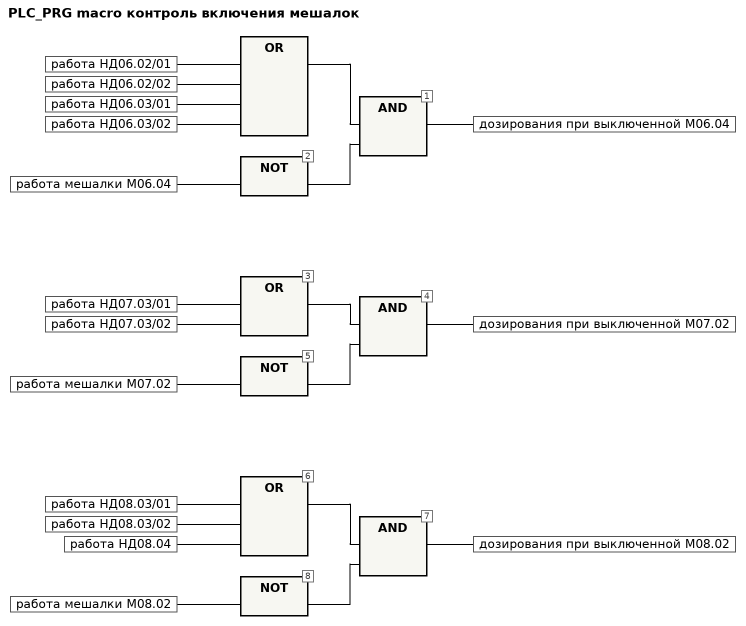
[picture p24: PLC_PRG macro контроль включения мешалок (CFC)]
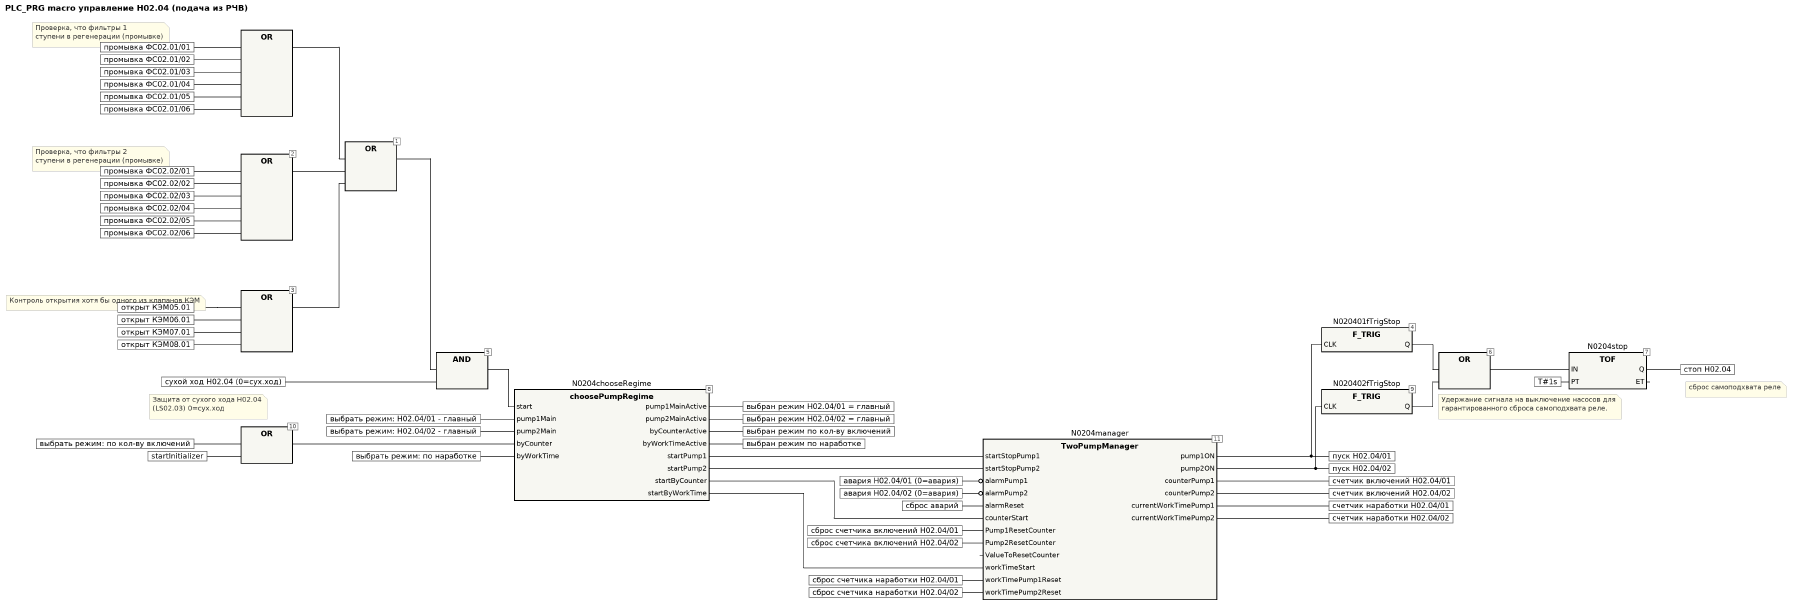
_CFC_ (* Continuous Function Chart, elements in execution order *)
(* Пуск Н02.04/02 *)
(* Пуск Н02.04/01 *)
(* Стоп Н02.04 *)
(* Сухой ход Н02.04 (LS02.03) 0=сух.ход *)
(* Клапан КЭМ08.01 открыт. *)
(* Клапан КЭМ07.01 открыт. *)
(* Клапан КЭМ06.01 открыт. *)
(* Клапан КЭМ05.01 открыт. *)
(* промывка ФС02.02/01 *)
(* промывка ФС02.02/02 *)
(* промывка ФС02.02/03 *)
(* промывка ФС02.02/04 *)
(* промывка ФС02.02/05 *)
(* промывка ФС02.02/06 *)
(* Авария Н02.04/02 (0=авария) *)
(* Авария Н02.04/01 (0=авария) *)
(* импульсный расходомер *)
(* авария Н04.04/02, 0=авария *)
(* авария Н04.04/01, 0=авария *)
(* сухой ход Н04.04, 0=защита *)
(* авт.пуск Н04.04 *)
(* пуск Н04.04/01 *)
(* пуск Н04.04/02 *)
(* стоп Н04.04 *)
(* подающий насос ФПК работает *)
(* статус КШЭ04.01 закрыт *)
(* Закрыть КШЭ04.01 *)
(* статус КШЭ04.01 открыт *)
(* Открыть КШЭ04.01 *)
(* авария ФПК *)
(* Авария входа AI6 ПЛК, давл.ФПК *)
(* Давление на входе ФПК / 0...16 бар (мах допуст.10) *)
(* LSА02.01 Перелив РЧВ02.03 *)
(* авария питания ЗДЭ02.25 *)
(* термоконтакт Н01.05/02 *)
(* термоконтакт Н01.05/01 *)
(* Авария ЧРП Н01.05 *)
(* КМ3 питание насоса 2 *)
(* КМ2 питание насоса 1 *)
(* КМ1 питание ЧРП *)
(* Пуск  Н01.05 *)
(* время на создание потока *)
(* управление Н01.05 - поддержание заданного расхода по FT01.02 *)
(* Стоп  Н01.05 (сброс самоподхвата реле) *)
(* SA1 Ручной выбор Н01.05/02 = главный *)
(* SA1 Ручной выбор Н01.05/01 = главный *)
(* LS01.04 - нижний уровень ОГМ01.04, сухой ход Н01.05 *)
(* LS01.03 - рабочий верхний уровень ОГМ01.04 автоматический пуск 01.05 *)
(* Статус ПУСК ЧРП Н01.05 *)
(* Инициализирует требуемые булевые переменные / в момент старта выполнения программы. *)
(* LSA01.02 перелив ОГМ01.04 *)
(* сухой ход НД08.03/02 *)
(* сухой ход НД08.03/01 *)
(* сухой ход НД08.03/02 *)
(* сухой ход НД08.03/01 *)
(* авария входа рН-метра QE01.02 *)
(* рН-метр QE01.01 на входе, / диапазон 0...14 *)
(* расходомер FT01.02 на входе, / диапазон 0...600куб/час *)
(* авария входа расходомера FT01.01 *)
(* управление 4...20мА НД08.04 *)
(* пуск/стоп НД08.04 *)
(* насос Н04.01 работает *)
(* авария НД08.04 *)
(* авария привода НД08.03/02 *)
(* авария привода НД08.03/01 *)
(* АВАРИИ *)
(* управление 4...20мА НД05.02/02 *)
(* пуск/стоп НД05.02/02 *)
(* авария НД05.02/02 *)
(* авария НД05.02/01 *)
(* пуск/стоп НД05.02/01 *)
(* управление 4...20мА НД05.02/01 *)
(* датчик температуры в помещении / (метран) диапазон: 0...+100С *)
(* лампа АВАРИЯ *)
(* авария входа датчика температуры *)
(* ошибка блока дозирования НД05.02 *)
(* авария НД06.02/02 *)
(* авария НД06.02/01 *)
(* управление 4...20мА НД06.02/02 *)
(* пуск/стоп НД06.02/02 *)
(* пуск/стоп НД06.02/01 *)
(* управление 4...20мА НД06.02/01 *)
(* авария НД06.03/02 *)
(* авария НД06.03/01 *)
(* управление 4...20мА НД06.03/02 *)
(* пуск/стоп НД06.03/02 *)
(* пуск/стоп НД06.03/01 *)
(* управление 4...20мА НД06.03/01 *)
(* авария НД05.02/02 *)
(* авария НД05.02/01 *)
(* авария НД06.02/02 *)
(* авария НД06.02/01 *)
(* авария НД06.03/02 *)
(* авария НД06.03/01 *)
(* авария НД07.03/02 *)
(* авария НД07.03/01 *)
(* пуск/стоп НД07.03/02 *)
(* пуск/стоп НД07.03/01 *)
(* управление 4...20мА НД07.03/02 *)
(* управление 4...20мА НД07.03/01 *)
(* авария НД07.03/02 *)
(* авария НД07.03/01 *)
(* авария привода НД08.03/02 *)
(* авария привода НД08.03/01 *)
(* управление 4...20мА НД08.03/02 *)
(* пуск/стоп НД08.03/02 *)
(* пуск/стоп НД08.03/01 *)
(* управление 4...20мА НД08.03/01 *)
(* авария НД08.04 *)
(* расходомер FT01.01 на входе, / диапазон 0...600куб/час *)
(* авария входа расходомера FT01.02 *)
(* авария входа рН-метра QE01.01 *)
(* рН-метр QE01.02 на входе, / диапазон 0...14 *)
(* статус ЗДЭ02.25 закрыт *)
(* LS02.02 Раб.верх.уровень РЧВ02.03 *)
(* Закрыть ЗДЭ02.25 *)
(* статус ЗДЭ02.25 открыт *)
(* LSА02.01 Перелив РЧВ02.03 *)
(* Открыть ЗДЭ02.25 *)
(* ФПК не запустился *)
(* ФПК готов к приему *)
(* подающий насос ФПК работает *)
(* авария ФПК *)
(* Давление на входе ФПК (0...16 бар) *)
(* датчик уровня осадка *)
(* Защита от сухого хода насоса ФПК *)
(* запуск фильтрации *)
(* время работы ФПК после спада сигнала датч.осадка *)
(* время контроля старта ФПК (по умолч.=3мин) *)
(* авария Н04.04/02 *)
(* авария Н04.04/01 *)
(* УФО вкл вручную без потока *)
(* авария УФО03.01/01 *)
(* авария УФО03.01/02 *)
(* авт.пускУФО03.01/01 *)
(* работа УФО03.01/01 *)
(* Для подачи предостережения на пульте / оператора (при необходимости), а также / сигнализации лампой АВАРИЯ. *)
(* авт.пускУФО03.01/02 *)
(* авария УФО03.01/01 *)
(* работа УФО03.01/02 *)
(* авария УФО03.01/02 *)
(* Контроль, если УФО включили вручную, / а потока при этом нет. *)
(* работа М06.04 (УПК) *)
(* работа М07.02 (УПЩ) *)
(* работа М08.02 (УПФ) *)
(* авария М06.04 (УПК) *)
(* авария М07.02 (УПЩ) *)
(* авария М08.02 (УПФ) *)
(* пуск/стоп НД07.03/02 *)
(* пуск/стоп НД07.03/01 *)
(* пуск/стоп НД08.04 *)
(* пуск/стоп НД06.02/02 *)
(* пуск/стоп НД06.02/01 *)
(* пуск/стоп НД06.03/02 *)
(* пуск/стоп НД06.03/01 *)
(* пуск/стоп НД08.03/02 *)
(* пуск/стоп НД08.03/01 *)
(* Авария Н02.04/02 (0=авария) *)
(* Защита от сухого хода Н02.04 / (LS02.03) 0=сух.ход *)
(* Авария Н02.04/01 (0=авария) *)
(* Стоп Н02.04 *)
(* Пуск Н02.04/02 *)
(* Пуск Н02.04/01 *)
(* Контроль открытия хотя бы одного из клапанов КЭМ *)
(* Клапан КЭМ08.01 открыт. *)
(* Клапан КЭМ07.01 открыт. *)
(* Клапан КЭМ06.01 открыт. *)
(* Клапан КЭМ05.01 открыт. *)
(* Удержание сигнала на выключение насосов для / гарантированного сброса самоподхвата реле. *)
(* промывка ФС02.02/01 *)
(* Проверка, что фильтры 2 / ступени в регенерации (промывке) *)
(* промывка ФС02.02/02 *)
(* промывка ФС02.02/03 *)
(* промывка ФС02.02/04 *)
(* промывка ФС02.02/05 *)
(* промывка ФС02.02/06 *)
(* промывка ФС02.01/01 *)
(* Проверка, что фильтры 1 / ступени в регенерации (промывке) *)
(* промывка ФС02.01/02 *)
(* промывка ФС02.01/03 *)
(* промывка ФС02.01/04 *)
(* промывка ФС02.01/05 *)
(* промывка ФС02.01/06 *)
(* промывка ФС02.01/01 *)
(* промывка ФС02.01/02 *)
(* промывка ФС02.01/03 *)
(* промывка ФС02.01/04 *)
(* промывка ФС02.01/05 *)
(* промывка ФС02.01/06 *)
(* Авария Н02.04/02 (0=авария) *)
(* Авария Н02.04/01 (0=авария) *)
#0 rTrigStartInitializer:R_TRIG(CLK: TRUE)
#1 startInitializer <= #0.Q
#2 MACRO контроль аналогового входа DD1_AI1(pin 1 "вход": DD1_AI1)
	(* Не смотрим конкретную ошибку, / определяем,что вход неисправен без расшифровки. *)
	#3 DD1_AI1_FT0101:DECODE_FLOAT(VALUE: pin 1, DEF_VALUE: -)
	#4 NE(#3._ERR, 0)
	out 2 "авария" <= #4
	out 1 "выход" <= #3.OUT_VALUE
END_MACRO
#5 DD1_AI1_FT0101value <= #2.out 1
#6 DD1_AI1_error <= #2.out 2
#7 MACRO контроль аналогового входа DD1_AI2(pin 1 "вход": DD1_AI2)
	(* Не смотрим конкретную ошибку, / определяем,что вход неисправен без расшифровки. *)
	#8 DD1_AI2_FT0102:DECODE_FLOAT(VALUE: pin 1, DEF_VALUE: -)
	#9 NE(#8._ERR, 0)
	out 2 "авария" <= #9
	out 1 "выход" <= #8.OUT_VALUE
END_MACRO
#10 DD1_AI2_FT0102value <= #7.out 1
#11 DD1_AI2_error <= #7.out 2
#12 MACRO контроль аналогового входа DD1_AI3(pin 1 "вход": DD1_AI3)
	(* Не смотрим конкретную ошибку, / определяем,что вход неисправен без расшифровки. *)
	#13 DD1_AI3_QE0101:DECODE_FLOAT(VALUE: pin 1, DEF_VALUE: -)
	#14 NE(#13._ERR, 0)
	out 2 "авария" <= #14
	out 1 "выход" <= #13.OUT_VALUE
END_MACRO
#15 DD1_AI3_QE0101value <= #12.out 1
#16 DD1_AI3_error <= #12.out 2
#17 OR(DD1_AI0_error, alarmHighTemperature, alarmLowTemperature, ND0502dosingError, NOT DD6_DI.0, NOT DD6_DI.1, ND0502dosingError, NOT DD6_DI.2, NOT DD6_DI.3, ND0602dosingError, NOT DD6_DI.4, NOT DD6_DI.5, ND0603dosingError, NOT DD6_DI.6, NOT DD6_DI.7, ND0803dosingError, NOT DD5_DI.12, NOT DD5_DI.13, DD1_DI6, DD1_DI7, NOT DD6_DI.16, ND0804dosingError, DD1_AI1_error, DD1_AI2_error, DD1_AI3_error, DD1_AI4_error, NOT DD6_DI.11, N010501alarm, N010502alarm, NOT DD9_DI.28, ZDE0225errorToOpen, ZDE0225errorToClose, NOT DD6_DI.13, DD1_AI5_error, DD7_DI.14, FPKnotStarted, FPKneedToClean, FPKkshe0401errorToOpen, FPKkshe0401errorToClose, NOT DD5_DI.14, NOT DD5_DI.15, DD5_DI.27, DD5_DI.29, UFO0301noFlowAttention, NOT DD5_DI.20, NOT DD5_DI.22, NOT DD5_DI.24, NOT DD5_DI.7, NOT DD5_DI.8)
#18 DD1_DO11 <= #17
#19 MACRO управление НД06.02 УПК(pin 1 "вход расходомера в куб/час": DD1_AI2_FT0102value, pin 2 "max производительность НД в мл/мин": ND0602setMaxDosVal, pin 3 "задание дозирования в мл/куб": ND0602setKoefProp, pin 4 "режим:1 насос главный": ND0602regimeP1M, pin 5 "режим: 2 насос главный": ND0602regimeP2M, pin 6 "режим: по наработке": ND0602regimeByWT, pin 7 "режим: по кол-ву включений": ND0602regimeByC, pin 8 "авария 1 насоса": DD6_DI.2, pin 9 "авария 2 насоса": DD6_DI.3, pin 10 "сброс аварий": alarmReset, pin 11 "сброс счетчика включений 1 насоса": ND0602resetCountP1, pin 12 "сброс ссчетчика включений 2 насоса": ND0602resetCountP2, pin 13 "сброс наработки 1 насоса": ND0602resetWorkTimeP1, pin 14 "сброс наработки 2 насоса": ND0602resetWorkTimeP2)
	(* Если на входе SEL = TRUE, / то нижнее значение, / иначе - то,что посередине. *)
	(* сигнал 4...20мА на НД06.02/01 *)
	(* сигнал 4...20мА на НД06.02/02 *)
	#20 SEL(#27.pump1ON, 0, #22.outputValue)
	#21 REAL_TO_WORD(#20)
	out 6 "выход 4...20мА насоса 1" <= #21
	#22 ND0602dosing:DosingPumpProportional(flowValue: pin 1, setMinPumpDosingValue: -, setMaxPumpDosingValue: pin 2, minOutputValue: -, maxOutputValue: -, setKoeffProportionality: pin 3, minFlowToStart: -)
	out 1 "ошибка блока дозирования" <= #22.dosingError
	#23 SEL(#27.pump2ON, 0, #22.outputValue)
	#24 REAL_TO_WORD(#23)
	out 7 "выход 4...20мА насоса 2" <= #24
	#25 ND0602regime:choosePumpRegime(start: #22.startDosingPump, pump1Main: pin 4, pump2Main: pin 5, byCounter: #26, byWorkTime: pin 6)
	out 2 "статус: 1 насос главный" <= #25.pump1MainActive
	out 3 "статус: 2 насос главный" <= #25.pump2MainActive
	out 4 "статус: по кол-ву включений" <= #25.byCounterActive
	#26 OR(pin 7, startInitializer)
	out 5 "статус: по наработке" <= #25.byWorkTimeActive
	#27 ND0602manager:TwoPumpManager(startStopPump1: #25.startPump1, startStopPump2: #25.startPump2, alarmPump1: #28, alarmPump2: #29, alarmReset: pin 10, counterStart: #25.startByCounter, Pump1ResetCounter: pin 11, Pump2ResetCounter: pin 12, ValueToResetCounter: -, workTimeStart: #25.startByWorkTime, workTimePump1Reset: pin 13, workTimePump2Reset: pin 14)
	out 12 "сигнал на включение насоса 1" <= #27.pump1ON
	#28 NOT(pin 8)
	out 13 "сигнал на включение насоса 2" <= #27.pump2ON
	out 8 "счетчик включений насоса 1" <= #27.counterPump1
	#29 NOT(pin 9)
	out 9 "счетчик включений насоса 2" <= #27.counterPump2
	out 10 "счетчик наработки насоса 1" <= #27.currentWorkTimePump1
	out 11 "счетчик наработки насоса 2" <= #27.currentWorkTimePump2
END_MACRO
#30 ND0602dosingError <= #19.out 1
#31 ND0602statRegimeP1M <= #19.out 2
#32 ND0602statRegimeP2M <= #19.out 3
#33 ND0602statRegimeByC <= #19.out 4
#34 ND0602statRegimeByWT <= #19.out 5
#35 DD10_AO1 <= #19.out 6
#36 DD10_AO2 <= #19.out 7
#37 ND0602counterP1 <= #19.out 8
#38 ND0602counterP2 <= #19.out 9
#39 ND0602workTimeP1 <= #19.out 10
#40 ND0602workTimeP2 <= #19.out 11
#41 DD4_DO.6 <= #19.out 12
#42 DD4_DO.7 <= #19.out 13
#43 MACRO контроль аналогового входа DD1_AI4(pin 1 "вход": DD1_AI4)
	(* Не смотрим конкретную ошибку, / определяем,что вход неисправен без расшифровки. *)
	#44 DD1_AI4_QE0102:DECODE_FLOAT(VALUE: pin 1, DEF_VALUE: -)
	#45 NE(#44._ERR, 0)
	out 2 "авария" <= #45
	out 1 "выход" <= #44.OUT_VALUE
END_MACRO
#46 DD1_AI4_QE0102value <= #43.out 1
#47 DD1_AI4_error <= #43.out 2
#48 MACRO управление НД05.02 УПГ(pin 1 "вход расходомера в куб/час": DD1_AI1_FT0101value, pin 2 "max производительность НД в мл/мин": ND0502setMaxDosVal, pin 3 "задание дозирования в мл/куб": ND0502setKoefProp, pin 4 "режим:1 насос главный": ND0502regimeP1M, pin 5 "режим: 2 насос главный": ND0502regimeP2M, pin 6 "режим: по наработке": ND0502regimeByWT, pin 7 "режим: по кол-ву включений": ND0502regimeByC, pin 8 "авария 1 насоса": DD6_DI.0, pin 9 "авария 2 насоса": DD6_DI.1, pin 10 "сброс аварий": alarmReset, pin 11 "сброс счетчика включений 1 насоса": ND0502resetCountP1, pin 12 "сброс ссчетчика включений 2 насоса": ND0502resetCountP2, pin 13 "сброс наработки 1 насоса": ND0502resetWorkTimeP1, pin 14 "сброс наработки 2 насоса": ND0502resetWorkTimeP2)
	(* Если на входе SEL = TRUE, / то нижнее значение, / иначе - то,что посередине. *)
	(* сигнал 4...20мА на НД05.02/01 *)
	(* сигнал 4...20мА на НД05.02/02 *)
	#49 SEL(#55.pump1ON, 0, #50.outputValue)
	out 6 "выход 4...20мА насоса 1" <= #49
	#50 ND0502dosing:DosingPumpProportional(flowValue: pin 1, setMinPumpDosingValue: -, setMaxPumpDosingValue: pin 2, minOutputValue: -, maxOutputValue: -, setKoeffProportionality: pin 3, minFlowToStart: -)
	out 1 "ошибка блока дозирования" <= #50.dosingError
	#51 SEL(#55.pump2ON, 0, #50.outputValue)
	#52 REAL_TO_WORD(#51)
	out 7 "выход 4...20мА насоса 2" <= #52
	#53 ND0502regime:choosePumpRegime(start: #50.startDosingPump, pump1Main: pin 4, pump2Main: pin 5, byCounter: #54, byWorkTime: pin 6)
	out 2 "статус: 1 насос главный" <= #53.pump1MainActive
	out 3 "статус: 2 насос главный" <= #53.pump2MainActive
	out 4 "статус: по кол-ву включений" <= #53.byCounterActive
	#54 OR(pin 7, startInitializer)
	out 5 "статус: по наработке" <= #53.byWorkTimeActive
	#55 ND0502manager:TwoPumpManager(startStopPump1: #53.startPump1, startStopPump2: #53.startPump2, alarmPump1: #56, alarmPump2: #57, alarmReset: pin 10, counterStart: #53.startByCounter, Pump1ResetCounter: pin 11, Pump2ResetCounter: pin 12, ValueToResetCounter: -, workTimeStart: #53.startByWorkTime, workTimePump1Reset: pin 13, workTimePump2Reset: pin 14)
	out 12 "сигнал на включение насоса 1" <= #55.pump1ON
	#56 NOT(pin 8)
	out 13 "сигнал на включение насоса 2" <= #55.pump2ON
	out 8 "счетчик включений насоса 1" <= #55.counterPump1
	#57 NOT(pin 9)
	out 9 "счетчик включений насоса 2" <= #55.counterPump2
	out 10 "счетчик наработки насоса 1" <= #55.currentWorkTimePump1
	out 11 "счетчик наработки насоса 2" <= #55.currentWorkTimePump2
END_MACRO
#58 ND0502dosingError <= #48.out 1
#59 ND0502statRegimeP1M <= #48.out 2
#60 ND0502statRegimeP2M <= #48.out 3
#61 ND0502statRegimeByC <= #48.out 4
#62 ND0502statRegimeByWT <= #48.out 5
#63 DD1_AO3 <= #48.out 6
#64 DD10_AO0 <= #48.out 7
#65 ND0502counterP1 <= #48.out 8
#66 ND0502counterP2 <= #48.out 9
#67 ND0502workTimeP1 <= #48.out 10
#68 ND0502workTimeP2 <= #48.out 11
#69 DD4_DO.4 <= #48.out 12
#70 DD4_DO.5 <= #48.out 13
#71 MACRO управление НД06.03 УПК(pin 1 "вход расходомера в куб/час": DD1_AI1_FT0101value, pin 2 "max производительность НД в мл/мин": ND0603setMaxDosVal, pin 3 "задание дозирования в мл/куб": ND0603setKoefProp, pin 4 "режим:1 насос главный": ND0603regimeP1M, pin 5 "режим: 2 насос главный": ND0603regimeP2M, pin 6 "режим: по наработке": ND0603regimeByWT, pin 7 "режим: по кол-ву включений": ND0603regimeByC, pin 8 "авария 1 насоса": DD6_DI.4, pin 9 "авария 2 насоса": DD6_DI.5, pin 10 "сброс аварий": alarmReset, pin 11 "сброс счетчика включений 1 насоса": ND0603resetCountP1, pin 12 "сброс ссчетчика включений 2 насоса": ND0603resetCountP2, pin 13 "сброс наработки 1 насоса": ND0603resetWorkTimeP1, pin 14 "сброс наработки 2 насоса": ND0603resetWorkTimeP2)
	(* Если на входе SEL = TRUE, / то нижнее значение, / иначе - то,что посередине. *)
	(* сигнал 4...20мА на НД06.03/01 *)
	(* сигнал 4...20мА на НД06.03/02 *)
	#72 SEL(#79.pump1ON, 0, #74.outputValue)
	#73 REAL_TO_WORD(#72)
	out 6 "выход 4...20мА насоса 1" <= #73
	#74 ND0603dosing:DosingPumpProportional(flowValue: pin 1, setMinPumpDosingValue: -, setMaxPumpDosingValue: pin 2, minOutputValue: -, maxOutputValue: -, setKoeffProportionality: pin 3, minFlowToStart: -)
	out 1 "ошибка блока дозирования" <= #74.dosingError
	#75 SEL(#79.pump2ON, 0, #74.outputValue)
	#76 REAL_TO_WORD(#75)
	out 7 "выход 4...20мА насоса 2" <= #76
	#77 ND0603regime:choosePumpRegime(start: #74.startDosingPump, pump1Main: pin 4, pump2Main: pin 5, byCounter: #78, byWorkTime: pin 6)
	out 2 "статус: 1 насос главный" <= #77.pump1MainActive
	out 3 "статус: 2 насос главный" <= #77.pump2MainActive
	out 4 "статус: по кол-ву включений" <= #77.byCounterActive
	#78 OR(pin 7, startInitializer)
	out 5 "статус: по наработке" <= #77.byWorkTimeActive
	#79 ND0603manager:TwoPumpManager(startStopPump1: #77.startPump1, startStopPump2: #77.startPump2, alarmPump1: #80, alarmPump2: #81, alarmReset: pin 10, counterStart: #77.startByCounter, Pump1ResetCounter: pin 11, Pump2ResetCounter: pin 12, ValueToResetCounter: -, workTimeStart: #77.startByWorkTime, workTimePump1Reset: pin 13, workTimePump2Reset: pin 14)
	out 12 "сигнал на включение насоса 1" <= #79.pump1ON
	#80 NOT(pin 8)
	out 13 "сигнал на включение насоса 2" <= #79.pump2ON
	out 8 "счетчик включений насоса 1" <= #79.counterPump1
	#81 NOT(pin 9)
	out 9 "счетчик включений насоса 2" <= #79.counterPump2
	out 10 "счетчик наработки насоса 1" <= #79.currentWorkTimePump1
	out 11 "счетчик наработки насоса 2" <= #79.currentWorkTimePump2
END_MACRO
#82 ND0603dosingError <= #71.out 1
#83 ND0603statRegimeP1M <= #71.out 2
#84 ND0603statRegimeP2M <= #71.out 3
#85 ND0603statRegimeByC <= #71.out 4
#86 ND0603statRegimeByWT <= #71.out 5
#87 DD10_AO3 <= #71.out 6
#88 DD10_AO4 <= #71.out 7
#89 ND0603counterP1 <= #71.out 8
#90 ND0603counterP2 <= #71.out 9
#91 ND0603workTimeP1 <= #71.out 10
#92 ND0603workTimeP2 <= #71.out 11
#93 DD4_DO.8 <= #71.out 12
#94 DD4_DO.9 <= #71.out 13
#95 MACRO управление НД08.03 УПФ(pin 1 "вход расходомера в куб/час": DD1_AI1_FT0101value, pin 2 "max производительность НД в мл/мин": ND0803setMaxDosVal, pin 3 "задание дозирования в мл/куб": ND0803setKoefProp, pin 4 "режим:1 насос главный": ND0803regimeP1M, pin 5 "режим: 2 насос главный": ND0803regimeP2M, pin 6 "режим: по наработке": ND0803regimeByWT, pin 7 "режим: по кол-ву включений": ND0803regimeByC, pin 8 "авария 1 насоса": DD5_DI.12, pin 9 "авария 2 насоса": DD5_DI.13, pin 10 "сброс аварий": alarmReset, pin 11 "сброс счетчика включений 1 насоса": ND0803resetCountP1, pin 12 "сброс ссчетчика включений 2 насоса": ND0803resetCountP2, pin 13 "сброс наработки 1 насоса": ND0803resetWorkTimeP1, pin 14 "сброс наработки 2 насоса": ND0803resetWorkTimeP2, pin 15 "сухой ход 1 насоса": DD1_DI6, pin 16 "сухой ход 2 насоса": DD1_DI7)
	(* Если на входе SEL = TRUE, / то нижнее значение, / иначе - то,что посередине. *)
	(* сигнал 4...20мА на НД08.03/01 *)
	(* сигнал 4...20мА на НД08.03/02 *)
	#96 SEL(#105.pump1ON, 0, #97.outputValue)
	out 6 "выход 4...20мА насоса 1" <= #96
	#97 ND0803dosing:DosingPumpProportional(flowValue: pin 1, setMinPumpDosingValue: -, setMaxPumpDosingValue: pin 2, minOutputValue: -, maxOutputValue: -, setKoeffProportionality: pin 3, minFlowToStart: -)
	out 1 "ошибка блока дозирования" <= #97.dosingError
	#98 SEL(#105.pump2ON, 0, #97.outputValue)
	out 7 "выход 4...20мА насоса 2" <= #98
	#99 ND0803regime:choosePumpRegime(start: #97.startDosingPump, pump1Main: pin 4, pump2Main: pin 5, byCounter: #100, byWorkTime: pin 6)
	out 2 "статус: 1 насос главный" <= #99.pump1MainActive
	out 3 "статус: 2 насос главный" <= #99.pump2MainActive
	out 4 "статус: по кол-ву включений" <= #99.byCounterActive
	#100 OR(pin 7, startInitializer)
	out 5 "статус: по наработке" <= #99.byWorkTimeActive
	out 12 "сигнал на включение насоса 1" <= #105.pump1ON
	#101 NOT(pin 8)
	#102 OR(#101, pin 15)
	out 13 "сигнал на включение насоса 2" <= #105.pump2ON
	#103 NOT(pin 9)
	#104 OR(#103, pin 16)
	#105 ND0803manager:TwoPumpManager(startStopPump1: #99.startPump1, startStopPump2: #99.startPump2, alarmPump1: #102, alarmPump2: #104, alarmReset: pin 10, counterStart: #99.startByCounter, Pump1ResetCounter: pin 11, Pump2ResetCounter: pin 12, ValueToResetCounter: -, workTimeStart: #99.startByWorkTime, workTimePump1Reset: pin 13, workTimePump2Reset: pin 14)
	out 8 "счетчик включений насоса 1" <= #105.counterPump1
	out 9 "счетчик включений насоса 2" <= #105.counterPump2
	out 10 "счетчик наработки насоса 1" <= #105.currentWorkTimePump1
	out 11 "счетчик наработки насоса 2" <= #105.currentWorkTimePump2
END_MACRO
#106 ND0803dosingError <= #95.out 1
#107 ND0803statRegimeP1M <= #95.out 2
#108 ND0803statRegimeP2M <= #95.out 3
#109 ND0803statRegimeByC <= #95.out 4
#110 ND0803statRegimeByWT <= #95.out 5
#111 DD1_AO1 <= #95.out 6
#112 DD1_AO2 <= #95.out 7
#113 ND0803counterP1 <= #95.out 8
#114 ND0803counterP2 <= #95.out 9
#115 ND0803workTimeP1 <= #95.out 10
#116 ND0803workTimeP2 <= #95.out 11
#117 DD1_DO3 <= #95.out 12
#118 DD1_DO4 <= #95.out 13
#119 MACRO управление НД07.03 УПЩ (поддержка рН, ПИД-регулятор)(pin 1 "вход рН-метра QE01.01": DD1_AI3_QE0101value, pin 2 "уставка рН": ND0703pHsetValue, pin 3 "режим:1 насос главный": ND0703regimeP1M, pin 4 "режим: 2 насос главный": ND0703regimeP2M, pin 5 "режим: по наработке": ND0703regimeByWT, pin 6 "режим: по кол-ву включений": ND0703regimeByC, pin 7 "авария 1 насоса": DD6_DI.6, pin 8 "авария 2 насоса": DD6_DI.7, pin 9 "сброс аварий": alarmReset, pin 10 "сброс счетчика включений 1 насоса": ND0703resetCountP1, pin 11 "сброс счетчика включений 2 насоса": ND0703resetCountP2, pin 12 "сброс наработки 1 насоса": ND0703resetWorkTimeP1, pin 13 "сброс наработки 2 насоса": ND0703resetWorkTimeP2, pin 14 "ручное управл.выходом Y (4...20мА)": ND0703YoutManual, pin 15 "1=ручное/0=автомат.управл.": ND0703YmanAuto, pin 16 "вход расходомера FT01.01 (куб.м/час)": DD1_AI1_FT0101value, pin 17 "коэфф.I": ND0703koeffI, pin 18 "коэфф.D": ND0703koeffD, pin 19 "коэфф.Р": ND0703koeffP)
	(* min расход в кубометрах в час / для неачала дозирования. *)
	(* Если на входе SEL = TRUE, / то нижнее значение, / иначе - то,что посередине. *)
	(* сигнал 4...20мА на НД07.03/01 *)
	(* сигнал 4...20мА на НД07.03/02 *)
	#120 ND0703pidReg:PID(ACTUAL: pin 1, SET_POINT: pin 2, KP: pin 19, TN: pin 17, TV: pin 18, Y_MANUAL: pin 14, Y_OFFSET: 12, Y_MIN: 4, Y_MAX: 20, MANUAL: pin 15, RESET: #120.OVERFLOW)
	#121 SEL(#128.pump1ON, 0, #120.Y)
	#122 REAL_TO_WORD(#121)
	out 5 "выход 4...20мА насоса 1" <= #122
	#123 SEL(#128.pump2ON, 0, #120.Y)
	#124 REAL_TO_WORD(#123)
	out 6 "выход 4...20мА насоса 2" <= #124
	#125 GE(pin 16, 10)
	#126 ND0703regime:choosePumpRegime(start: #125, pump1Main: pin 3, pump2Main: pin 4, byCounter: #127, byWorkTime: pin 5)
	out 1 "статус: 1 насос главный" <= #126.pump1MainActive
	out 2 "статус: 2 насос главный" <= #126.pump2MainActive
	out 3 "статус: по кол-ву включений" <= #126.byCounterActive
	out 4 "статус: по наработке" <= #126.byWorkTimeActive
	#127 OR(pin 6, startInitializer)
	#128 ND0703manager:TwoPumpManager(startStopPump1: #126.startPump1, startStopPump2: #126.startPump2, alarmPump1: #129, alarmPump2: #130, alarmReset: pin 9, counterStart: #126.startByCounter, Pump1ResetCounter: pin 10, Pump2ResetCounter: pin 11, ValueToResetCounter: -, workTimeStart: #126.startByWorkTime, workTimePump1Reset: pin 12, workTimePump2Reset: pin 13)
	out 11 "сигнал на включение насоса 1" <= #128.pump1ON
	#129 NOT(pin 7)
	out 12 "сигнал на включение насоса 2" <= #128.pump2ON
	out 7 "счетчик включений насоса 1" <= #128.counterPump1
	#130 NOT(pin 8)
	out 8 "счетчик включений насоса 2" <= #128.counterPump2
	out 9 "счетчик наработки насоса 1" <= #128.currentWorkTimePump1
	out 10 "счетчик наработки насоса 2" <= #128.currentWorkTimePump2
END_MACRO
#131 ND0703statRegimeP1M <= #119.out 1
#132 ND0703statRegimeP2M <= #119.out 2
#133 ND0703statRegimeByC <= #119.out 3
#134 ND0703statRegimeByWT <= #119.out 4
#135 DD10_AO5 <= #119.out 5
#136 DD10_AO6 <= #119.out 6
#137 ND0703counterP1 <= #119.out 7
#138 ND0703counterP2 <= #119.out 8
#139 ND0703workTimeP1 <= #119.out 9
#140 ND0703workTimeP2 <= #119.out 10
#141 DD4_DO.10 <= #119.out 11
#142 DD4_DO.11 <= #119.out 12
#143 MACRO управление НД08.04 УПФ(pin 1 "насос Н04.01 работает": DD7_DI.13, pin 2 "авария НД08.04": DD6_DI.16, pin 3 "уставкаНД08.04(0...100%)": ND0804doseValue)
	(* Преобразует сигнал 0...100 / пропорционально в 4...20мА *)
	#144 AND(pin 1, pin 2)
	out 1 "пуск/стоп НД08.04" <= #144
	#145 ND0804linearTransformator:LIN_TRAFO(IN: pin 3, IN_MIN: 0, IN_MAX: 100, OUT_MIN: 4, OUT_MAX: 20)
	#146 REAL_TO_WORD(#145.OUT)
	out 2 "управление НД08.04 (4...20мА)" <= #146
	out 3 "ошибка блока дозирования" <= #145.ERROR
END_MACRO
#147 DD4_DO.12 <= #143.out 1
#148 DD10_AO7 <= #143.out 2
#149 ND0804dosingError <= #143.out 3
#150 MACRO контроль температуры в помещении(pin 1 "вход датчика температуры": DD1_AI0, pin 2 "минимально допустимая температура в помещении": maxTemperature, pin 3 "максимально допустимая температура в помещении": minTemperature)
	(* не смотрим конкретный тип ошибки / (работает не точно, обрыв определяет как слишком маленькое значение) / если не равно 0 - значит на входе ошибка *)
	(* задаем границы допустимой температуры в помещении / проверяем что измеренное значение в заданном диапазоне *)
	#151 DD1_AI0_temperature:DECODE_FLOAT(VALUE: pin 1, DEF_VALUE: -)
	#152 NE(#151._ERR, 0)
	out 2 "авария датчика температуры" <= #152
	out 1 "температура в помещении" <= #151.OUT_VALUE
	#153 REAL_TO_INT(#151.OUT_VALUE)
	#154 temperatureLimits:LIMITALARM(IN: #153, HIGH: pin 3, LOW: pin 2)
	out 3 "температура выше заданного диапазона" <= #154.O
	out 4 "температура ниже заданного диапазона" <= #154.U
	#155 temperatureLimits:LIMITALARM(IN: -, HIGH: -, LOW: -)
END_MACRO
#156 temperatureValue <= #150.out 1
#157 DD1_AI0_error <= #150.out 2
#158 alarmHighTemperature <= #150.out 3
#159 alarmLowTemperature <= #150.out 4
#160 MACRO контроль аналогового входа DD1_AI5(pin 1 "вход": DD1_AI5)
	(* Не смотрим конкретную ошибку, / определяем,что вход неисправен без расшифровки. *)
	#161 DD1_AI5_FPK:DECODE_FLOAT(VALUE: pin 1, DEF_VALUE: -)
	#162 NE(#161._ERR, 0)
	out 2 "авария" <= #162
	out 1 "выход" <= #161.OUT_VALUE
END_MACRO
#163 DD1_AI5_FPKpressureValue <= #160.out 1
#164 DD1_AI5_error <= #160.out 2
#165 MACRO управление Н01.05(pin 1 "статус ПУСК ЧРП (реле)": DD5_DI.4, pin 2 "LS01.03 раб.уров.": DD6_DI.12, pin 3 "LS01.04 ниж.уров.(сух.ход)": DD5_DI.0, pin 4 "SA1ручной выб.Н01.05/01-главный": DD5_DI.5, pin 5 "SA1ручной выб.Н01.05/02-главный": DD5_DI.6, pin 6 "включить режим "по кол.вкл."": N0105regimeByC, pin 7 "включить режим "по наработке"": N0105regimeByWT, pin 8 "значение расхода от FT01.02": DD1_AI2_FT0102value, pin 9 "уставка расхода": N0105flowSetValue, pin 10 "время на создание потока": N0105minFlowTime, pin 11 "Р-коэфф.": N0105koeffP, pin 12 "I-коэфф": N0105koeffI, pin 13 "Д-коэфф": N0105koeffD, pin 14 "управление ЧРП в ручн.реж.(4...20мА)": N0105YoutManual, pin 15 "переключатель управление ЧРП РУЧН/АВТ": N0105YmanAuto, pin 16 "мин.допустимый расход": N0105minFlow, pin 17 "термоконтакт Н01.05/01": DD5_DI.2, pin 18 "термоконтакт Н01.05/02": DD5_DI.3, pin 19 "авария ЧРП Н01.05": DD5_DI.1, pin 20 "сброс аварии": alarmReset, pin 21 "сброс кол-ва вкл.Н01.05/01": N0105resetCountP1, pin 22 "сброс кол-ва вкл.Н01.05/02": N0105resetCountP2, pin 23 "сброс наработки Н01.05/01": N0105resetWorkTimeP1, pin 24 "сброс наработки Н01.05/02": N0105resetWorkTimeP2)
	(* Если насос создает давление меньше / указанного, то авария. *)
	(* если на входе true / то нижнее значение, / иначе то, что посередине *)
	(* по умолчанию при старте программы *)
	(* управление Н01.05 - поддержание / заданного расхода по FT01.02 *)
	(* режимы по количеству включений,  или по наработке / активны если оба входа SA1 не активны *)
	(* Пуск  Н01.05 *)
	(* время на создание потока *)
	#166 OR(pin 2, #167.Q)
	#167 N0105startTrig:R_TRIG(CLK: pin 1)
	#168 N0105stopTrig:F_TRIG(CLK: pin 1)
	#169 N0105startTrigg:RS(SET: #166, RESET1: #171)
	#170 N0105regime:choosePumpRegime(start: #169.Q1, pump1Main: pin 4, pump2Main: pin 5, byCounter: #174, byWorkTime: #180)
	out 2 "статус режим "Н01.05/01 - главный"" <= #170.pump1MainActive
	out 3 "статус режим "Н01.05/02 - главный"" <= #170.pump2MainActive
	out 4 "статус режим "по кол-ву вкл."" <= #170.byCounterActive
	#171 OR(#168.Q, #172)
	out 5 "статус режим "по наработке"." <= #170.byWorkTimeActive
	#172 NOT(pin 3)
	#173 NOT(#169.Q1)
	out 1 "СТОП (сброс самоподхвата реле пуска ЧРП)." <= #173
	#174 AND(NOT pin 4, NOT pin 5, #177.Q1)
	#175 OR(pin 6, startInitializer)
	#176 N0105regByCinit:R_TRIG(CLK: #175)
	#177 N0105regByCtrig:RS(SET: #176.Q, RESET1: #185.Q)
	#178 N0105twoPumpOneDriveManager:TwoPumpOneDriveManager(startStopPump1: #170.startPump1, startStopPump2: #170.startPump2, alarmPump1: N010501alarm, alarmPump2: N010502alarm, alarmReset: alarmReset, counterStart: #170.startByCounter, Pump1ResetCounter: pin 21, Pump2ResetCounter: pin 22, ValueToResetCounter: -, workTimeStart: #170.startByWorkTime, workTimePump1Reset: pin 23, workTimePump2Reset: pin 24, timeKM1off: -, timeKM23DelayON: -, timeKM23offDelay: -, timeReadyToStartDelay: -)
	out 6 "кол-во включений Н01.05/01" <= #178.counterPump1
	#179 AND(#178.pump1active, #195)
	out 7 "кол-во включений Н01.05/02" <= #178.counterPump2
	out 8 "наработка Н01.05/01" <= #178.currentWorkTimePump1
	out 15 "авария Н01.05/01" <= #183.Q1
	#180 AND(NOT pin 4, NOT pin 5, #186.Q1)
	out 9 "наработка Н01.05/02" <= #178.currentWorkTimePump2
	out 10 "КМ1-питание ЧРП" <= #178.DriveKM
	#181 AND(#178.pump1active, #187)
	#182 OR(#179, #181)
	#183 N010501alarmTrig:RS(SET: #182, RESET1: pin 20)
	#184 N010501alarm <= #183.Q1
	#185 N0105regWTinit:R_TRIG(CLK: pin 7)
	#186 N0105regWTtrig:RS(SET: #185.Q, RESET1: #176.Q)
	out 11 "КМ2-питание Н01.05/01" <= #178.pump1KM
	out 12 "КМ3-питание Н01.05/02" <= #178.pump2KM
	#187 OR(NOT pin 17, NOT pin 19)
	out 13 "пуск ЧРП (Н01.05)" <= #178.driveStart
	#188 OR(NOT pin 19, NOT pin 18)
	out 16 "авария Н01.05/02" <= #191.Q1
	#189 AND(#188, #178.pump2active)
	#190 OR(#189, #193)
	#191 N010502alarmTrig:RS(SET: #190, RESET1: pin 20)
	#192 N010502alarm <= #191.Q1
	#193 AND(#178.pump2active, #195)
	#194 N0105timerminFlow:TON(IN: #178.driveStart, PT: pin 10)
	#195 AND(#194.Q, #196)
	#196 LE(pin 8, pin 16)
	#197 SEL(#178.driveStart, 0, #198.Y)
	out 14 "управление ЧРП (4...20мА)" <= #197
	#198 N0105pidReg:PID(ACTUAL: pin 8, SET_POINT: pin 9, KP: pin 11, TN: pin 12, TV: pin 13, Y_MANUAL: pin 14, Y_OFFSET: -, Y_MIN: 4, Y_MAX: 20, MANUAL: pin 15, RESET: #198.OVERFLOW)
END_MACRO
#199 DD4_DO.13 <= #165.out 1
#200 N0105statRegimeP1M <= #165.out 2
#201 N0105statRegimeP2M <= #165.out 3
#202 N0105statRegimeByC <= #165.out 4
#203 N0105statRegimeByWT <= #165.out 5
#204 N0105counterP1 <= #165.out 6
#205 N0105counterP2 <= #165.out 7
#206 N0105workTimeP1 <= #165.out 8
#207 N0105workTimeP2 <= #165.out 9
#208 DD2_DO.0 <= #165.out 10
#209 DD2_DO.1 <= #165.out 11
#210 DD2_DO.2 <= #165.out 12
#211 DD1_DO0 <= #165.out 13
#212 DD1_AO0 <= #165.out 14
#213 N010501alarm <= #165.out 15
#214 N010502alarm <= #165.out 16
#215 MACRO Сигналы работы с ФП04.02 (фильтр-пресс)(pin 1 "датчик уровня осадка": DD7_DI.15, pin 2 "время работы ФПК (после выкл.датч.осадка)": FPKtimeToWork, pin 3 "защита от сухого хода": DD6_DI.10, pin 4 "ошибка входа AI (обрыв)": DD1_AI5_error, pin 5 "авария ФПК": DD7_DI.14, pin 6 "фильтр-пресс готов к приему": DD7_DI.12, pin 7 "давление на входе в ФПК": DD1_AI5_FPKpressureValue, pin 8 "мах допустимое давление": FPKmaxPressureValue, pin 9 "подающий насос ФПК работает": DD7_DI.13, pin 10 "время контроля старта ФПК": FPKnotStartedTime, pin 11 "сброс аварий": alarmReset)
	(* Условие сброса сигнала л грязном фильтр-прессе: / 1. Пропал сигнал о готовности ФПК; / 2. Появился сигнал о готовности ФПК. / Это значит, что оператор раздвигал плиты, / чистил и снова сдвигал их. *)
	(* максимально допустимое давление / на входе ФПК *)
	(* Давление на входе ФПК / 0...16 бар (мах допуст.10) *)
	(* Время работы ФПК после / спада сигнала уровня осадка / по умолч.15мин. *)
	(* LES01.01-сигнал датчика уровня осадка ОГМ01.04 / запуск процесса фильтрации *)
	(* LS01.01-нижн.уровень на входе ОГМ01.04 / защита от сух. хода насоса ФПК *)
	(* ФПК готов к приему осадка *)
	#216 FPKneedToCleanResetFtrig:F_TRIG(CLK: FPKneedToCleanReset)
	#217 FPKstartTrig:RS(SET: pin 1, RESET1: #223)
	out 1 "запуск/старт ФПК" <= #217.Q1
	#218 FPKstopTimer:TOF(IN: pin 1, PT: pin 2)
	#219 FPKstopFtrig:F_TRIG(CLK: #218.Q)
	#220 AND(#217.Q1, #221)
	#221 NOT(pin 11)
	#222 AND(#217.Q1, #224.Q, #226)
	out 2 "ФПК не стартовал" <= #222
	#223 OR(#219.Q, pin 4, pin 5, #225, #227, #230.Q1)
	#224 FPKnotStartedTimer:TON(IN: #220, PT: pin 10)
	#225 NOT(pin 3)
	#226 NOT(pin 9)
	#227 NOT(pin 6)
	#228 AND(#217.Q1, #229)
	#229 GE(pin 7, pin 8)
	#230 FPKneedToCleanTrig:RS(SET: #228, RESET1: #216.Q)
	out 3 "ФПК нужно почистить!" <= #230.Q1
	#231 S FPKneedToCleanReset <= #230.Q1
	#232 FPKneedToCleanResetRtrig:R_TRIG(CLK: pin 6)
	#233 R FPKneedToCleanReset <= #232.Q
END_MACRO
#234 DD1_DO10 <= #215.out 1
#235 FPKnotStarted <= #215.out 2
#236 FPKneedToClean <= #215.out 3
#237 MACRO клапан шаровый перед ФПК (КШЭ04.01)(pin 1 "сигнал "подающий насос ФПК" работает": DD7_DI.13, pin 2 "статус КШЭ04.01 открыт": DD9_DI.2, pin 3 "статус КШЭ04.01 закрыт": DD9_DI.3, pin 4 "сброс аварий": alarmReset, pin 5 "время на открытие/закрытие": timeToOpenCloseValve)
	#238 FPKkshe0401DelayToOpen:TON(IN: #240.outputOpen, PT: T#1s)
	out 1 "выход на открытие КШЭ04.01" <= #238.Q
	#239 FPKkshe0401DelayToClose:TON(IN: #240.outputClose, PT: T#1s)
	out 2 "выход на закрытие КШЭ04.01" <= #239.Q
	#240 FPKkshe0401:SimpleValve(inputOpen: pin 1, inputClose: #241, statusOpen: pin 2, statusClose: pin 3, reset: pin 4, timeToOpenClose: pin 5)
	#241 NOT(pin 1)
	out 3 "авария на открытие КШЭ04.01" <= #240.errorToOpen
	out 4 "авария на закрытие КШЭ04.01" <= #240.errorToClose
END_MACRO
#242 DD4_DO.2 <= #237.out 1
#243 DD4_DO.3 <= #237.out 2
#244 FPKkshe0401errorToOpen <= #237.out 3
#245 FPKkshe0401errorToClose <= #237.out 4
#246 MACRO управление Н04.04 (дренажные)(pin 1 "защита от сухого хода Н04.04": DD5_DI.18, pin 2 "автоматич.пускН04.04": DD5_DI.19, pin 3 "режим Н04.04/01 главный": N0404regimeP1M, pin 4 "режим Н04.04/02 главный": N0404regimeP2M, pin 5 "режим по кол-ву включений": N0404regimeByC, pin 6 "режим по наработке": N0404regimeWT, pin 7 "авария Н04.04/01": DD5_DI.15, pin 8 "авария Н04.04/02": DD5_DI.14, pin 9 "сброс аварий": alarmReset, pin 10 "сброс счетчика включений Н04.04/01": N0404resetCountP1, pin 11 "сброс счетчика включений Н04.04/02": N0404resetCountP2, pin 12 "сброс счетчика наработки Н04.04/01": N0404resetWorkTimeP1, pin 13 "сброс счетчика наработки Н04.04/02": N0404resetWorkTimeP2)
	(* 0=авария *)
	(* сухой ход Н04.04 / 0=защита *)
	(* от поплавка *)
	(* насосы имеют электрическую блокировку / от одновременного включения *)
	(* Излишняя перестраховка по сухому ходу, / на уровне реле уже все отрабатывается. *)
	(* сбрасывает самоподхват пускового реле *)
	#247 NOT(pin 1)
	out 1 "стоп Н04.04" <= #247
	#248 AND(pin 1, pin 2)
	#249 N0401choosePumpRegime:choosePumpRegime(start: #248, pump1Main: pin 3, pump2Main: pin 4, byCounter: #250, byWorkTime: pin 6)
	out 2 "выбран режим: Н04.04/01 главный" <= #249.pump1MainActive
	out 3 "выбран режим: Н04.04/02 главный" <= #249.pump2MainActive
	out 4 "выбран режим: по кол-ву включений" <= #249.byCounterActive
	#250 OR(startInitializer, pin 5)
	out 5 "выбран режим: по наработке" <= #249.byWorkTimeActive
	#251 N0404twoPumpManager:TwoPumpManager(startStopPump1: #249.startPump1, startStopPump2: #249.startPump2, alarmPump1: #252, alarmPump2: #253, alarmReset: pin 9, counterStart: #249.startByCounter, Pump1ResetCounter: pin 10, Pump2ResetCounter: pin 11, ValueToResetCounter: -, workTimeStart: #249.startByWorkTime, workTimePump1Reset: pin 12, workTimePump2Reset: pin 13)
	out 6 "пуск Н04.04/01" <= #251.pump1ON
	#252 NOT(pin 7)
	out 7 "пуск Н04.04/02" <= #251.pump2ON
	out 8 "счетчик кол-ва включений Н04.04/01" <= #251.counterPump1
	#253 NOT(pin 8)
	out 9 "счетчик кол-ва включений Н04.04/02" <= #251.counterPump2
	out 10 "счетчик времени наработки Н04.04/01" <= #251.currentWorkTimePump1
	out 11 "счетчик времени наработки Н04.04/02" <= #251.currentWorkTimePump2
END_MACRO
#254 DD4_DO.15 <= #246.out 1
#255 N0404statRegimeP1M <= #246.out 2
#256 N0404statRegimeP2M <= #246.out 3
#257 N0404statRegimeByC <= #246.out 4
#258 N0404statRegimeWT <= #246.out 5
#259 DD1_DO5 <= #246.out 6
#260 DD1_DO6 <= #246.out 7
#261 N0404counterP1 <= #246.out 8
#262 N0404counterP2 <= #246.out 9
#263 N0404workTimeP1 <= #246.out 10
#264 N0404workTimeP2 <= #246.out 11
#265 MACRO Наполнение РЧВ02.03 (заслонка ЗДЭ02.25)(pin 1 "LS02.02раб.верх.уровень РЧВ": DD6_DI.14, pin 2 "LSA02.01 Перелив РЧВ": DD6_DI.13, pin 3 "статус ЗДЭ02.25 открыт": DD9_DI.0, pin 4 "статус ЗДЭ02.25 закрыт": DD9_DI.1, pin 5 "сброс аварий": alarmReset, pin 6 "время на открытие/закрытие": timeToOpenCloseValve)
	#266 NOT(pin 1)
	#267 ZDE0225:SimpleValve(inputOpen: pin 1, inputClose: #268, statusOpen: pin 3, statusClose: pin 4, reset: pin 5, timeToOpenClose: pin 6)
	out 1 "выход на открытие ЗДЭ02.25" <= #267.outputOpen
	#268 OR(#266, #269)
	out 2 "выход на закрытие ЗДЭ02.25" <= #267.outputClose
	out 3 "авария на открытие ЗДЭ02.25" <= #267.errorToOpen
	#269 NOT(pin 2)
	out 4 "авария на закрытие ЗДЭ02.25" <= #267.errorToClose
END_MACRO
#270 DD4_DO.0 <= #265.out 1
#271 DD4_DO.1 <= #265.out 2
#272 ZDE0225errorToOpen <= #265.out 3
#273 ZDE0225errorToClose <= #265.out 4
#274 MACRO Работа УФО03.01(pin 1 "Работа УФО03.01/01": DD5_DI.26, pin 2 "Работа УФО03.01/02": DD5_DI.28, pin 3 "Значение расхода от FT01.02": DD1_AI2_FT0102value, pin 4 "мин.допустимый расход для насосов Н01.05": N0105minFlow, pin 5 "Задержка включения УФО на создание потока": UFO0301startDelayTime, pin 6 "выбор режим: УФО03.01/01 главное": UFO0301regimeP1M, pin 7 "выбор режим: УФО03.01/02 главное": UFO0301regimeP2M, pin 8 "выбор режим: по кол-ву включений": UFO0301regimeByC, pin 9 "выбор режим: по наработке": UFO0301regimeWT, pin 10 "авария УФО03.01/01": DD5_DI.27, pin 11 "авария УФО03.01/02": DD5_DI.29, pin 12 "сброс аварий": alarmReset, pin 13 "сброс счетчика включений УФО03.01/01": UFO0301resetCountP1, pin 14 "сброс счетчика включений УФО03.01/02": UFO0301resetCountP2, pin 15 "сброс счетчика наработки УФО03.01/01": UFO0301resetWorkTimeP1, pin 16 "сброс счетчика наработки УФО03.01/02": UFO0301resetWorkTimeP2)
	(* Включаем УФО, если расходомер показывает расход больше, / чем заданный как минимально допустимый для работы насосов Н01.05. *)
	(* Задержка старта УФО *)
	(* Для подачи предостережения на пульте / оператора (при необходимости), а также / сигнализации лампой АВАРИЯ. *)
	(* Контроль, если УФО включили вручную, / а потока при этом нет. *)
	#275 OR(pin 1, pin 2)
	#276 AND(#275, #277)
	out 1 "УФО вкл без потока" <= #276
	#277 NOT(#279.Q)
	#278 GE(pin 3, pin 4)
	#279 UFO0301startDelay:TON(IN: #278, PT: pin 5)
	#280 UFO0301regimeManager:choosePumpRegime(start: #279.Q, pump1Main: pin 6, pump2Main: pin 7, byCounter: #281, byWorkTime: pin 9)
	out 2 "активен режим - главное УФО 03.01/01" <= #280.pump1MainActive
	out 3 "активен режим - главное УФО 03.01/02" <= #280.pump2MainActive
	out 4 "активен режим - по кол-ву включений" <= #280.byCounterActive
	#281 OR(startInitializer, pin 8)
	out 5 "активен режим - по наработке" <= #280.byWorkTimeActive
	#282 UFO0301manager:TwoPumpManager(startStopPump1: #280.startPump1, startStopPump2: #280.startPump2, alarmPump1: pin 10, alarmPump2: pin 11, alarmReset: pin 12, counterStart: #280.startByCounter, Pump1ResetCounter: pin 13, Pump2ResetCounter: pin 14, ValueToResetCounter: -, workTimeStart: #280.startByWorkTime, workTimePump1Reset: pin 15, workTimePump2Reset: pin 16)
	out 6 "авт. пуск УФО03.01/01" <= #282.pump1ON
	out 7 "авт. пуск УФО03.01/02" <= #282.pump2ON
	out 8 "счетчик включений УФО03.01/01" <= #282.counterPump1
	out 9 "счетчик включений УФО03.01/02" <= #282.counterPump2
	out 10 "счетчик наработки УФО03.01/01" <= #282.currentWorkTimePump1
	out 11 "счетчик наработки УФО03.01/02" <= #282.currentWorkTimePump2
END_MACRO
#283 UFO0301noFlowAttention <= #274.out 1
#284 UFO0301statRegimeP1M <= #274.out 2
#285 UFO0301statRegimeP2M <= #274.out 3
#286 UFO0301statRegimeByC <= #274.out 4
#287 UFO0301statRegimeWT <= #274.out 5
#288 DD1_DO8 <= #274.out 6
#289 DD1_DO9 <= #274.out 7
#290 UFO0301counterP1 <= #274.out 8
#291 UFO0301counterP2 <= #274.out 9
#292 UFO0301workTimeP1 <= #274.out 10
#293 UFO0301workTimeP2 <= #274.out 11
#294 MACRO импульсный счетчик FQS0301(pin 1 "вход от счетчика": DD6_DI.19, pin 2 "вес импульса счетчика": FQS0301impulsValue, pin 3 "сброс счетчика": FQS0301reset, pin 4 "величина коррекции счетчика": FQS0301correction, pin 5 "прибавить коррекцию": FQS0301addCorrection, pin 6 "вычесть коррекцию": FQS0301deleteCorrection)
	(* число, коорое будем прибавлять или / вычитать из накопленной суммы стоков. *)
	(* коррекция показаний счетчика. *)
	(* Если в результате коррекции накопленная сумма станет меньше нуля, то она принудительно станет равна нулю. *)
	(* значение в UDINT, целочисленное, / округляется по правилам арифметики. *)
	(* значение в REAL (в какой-то момент начинает / отображаться в экспоненциальной форме) *)
	(* сброс показаний счетчика *)
	#295 FQS0301rTrig:R_TRIG(CLK: pin 1)
	#296 ADD(EN: #295.Q, FQS0301totalAmount, pin 2)
	out 1 "накопленная сумма стоков (REAL)" <= #296
	#297 REAL_TO_UDINT(FQS0301totalAmount)
	out 2 "накопленная сумма стоков (UDINT)" <= #297
	#298 FQS0301resetRtrig:R_TRIG(CLK: pin 3)
	#299 MOVE(EN: #298.Q, 0)
	#300 FQS0301totalAmount <= #299
	#301 FQS0301addCorrRtrig:R_TRIG(CLK: pin 5)
	#302 ADD(EN: #301.Q, FQS0301totalAmount, pin 4)
	#303 FQS0301totalAmount <= #302
	#304 SUB(EN: #306.Q, FQS0301totalAmount, pin 4)
	#305 FQS0301totalAmount <= #304
	#306 FQS0301deleteCorrRtrig:R_TRIG(CLK: pin 6)
	#307 LT(FQS0301totalAmount, 0)
	#308 MOVE(EN: #307, 0)
	#309 FQS0301totalAmount <= #308
END_MACRO
#310 FQS0301totalAmount <= #294.out 1
#311 FQS0301totalAmountUDINT <= #294.out 2
#312 MACRO контроль включения мешалок(pin 1 "работа НД06.02/01": DD4_DO.6, pin 2 "работа НД06.02/02": DD4_DO.7, pin 3 "работа НД06.03/01": DD4_DO.8, pin 4 "работа НД06.03/02": DD4_DO.9, pin 5 "работа мешалки М06.04": DD5_DI.21, pin 6 "работа НД07.03/01": DD4_DO.10, pin 7 "работа НД07.03/02": DD4_DO.11, pin 8 "работа мешалки М07.02": DD5_DI.23, pin 9 "работа НД08.03/01": DD1_DO3, pin 10 "работа НД08.03/02": DD1_DO4, pin 11 "работа НД08.04": DD4_DO.12, pin 12 "работа мешалки М08.02": DD5_DI.25)
	#313 OR(pin 1, pin 2, pin 3, pin 4)
	#314 AND(#313, #315)
	out 1 "дозирования при выключенной М06.04" <= #314
	#315 NOT(pin 5)
	#316 OR(pin 6, pin 7)
	#317 AND(#316, #318)
	out 2 "дозирования при выключенной М07.02" <= #317
	#318 NOT(pin 8)
	#319 OR(pin 9, pin 10, pin 11)
	#320 AND(#319, #321)
	out 3 "дозирования при выключенной М08.02" <= #320
	#321 NOT(pin 12)
END_MACRO
#322 M0604attention <= #312.out 1
#323 M0702attention <= #312.out 2
#324 M0802attention <= #312.out 3
#325 MACRO управление Н02.04 (подача из РЧВ)(pin 1 "промывка ФС02.01/01": DD6_DI.20, pin 2 "промывка ФС02.01/02": DD6_DI.22, pin 3 "промывка ФС02.01/03": DD6_DI.24, pin 4 "промывка ФС02.01/04": DD6_DI.26, pin 5 "промывка ФС02.01/05": DD6_DI.28, pin 6 "промывка ФС02.01/06": DD6_DI.30, pin 7 "промывка ФС02.02/01": DD7_DI.0, pin 8 "промывка ФС02.02/02": DD7_DI.2, pin 9 "промывка ФС02.02/03": DD7_DI.4, pin 10 "промывка ФС02.02/04": DD7_DI.6, pin 11 "промывка ФС02.02/05": DD7_DI.8, pin 12 "промывка ФС02.02/06": DD7_DI.10, pin 13 "открыт КЭМ05.01": DD1_DI11, pin 14 "открыт КЭМ06.01": DD1_DI10, pin 15 "открыт КЭМ07.01": DD1_DI9, pin 16 "открыт КЭМ08.01": DD1_DI8, pin 17 "сухой ход Н02.04 (0=сух.ход)": DD5_DI.11, pin 18 "выбрать режим: Н02.04/01 - главный": N0204regimeP1M, pin 19 "выбрать режим: Н02.04/02 - главный": N0204regimeP2M, pin 20 "выбрать режим: по кол-ву включений": N0204regimeByC, pin 21 "выбрать режим: по наработке": N0204regimeWT, pin 22 "авария Н02.04/01 (0=авария)": DD5_DI.7, pin 23 "авария Н02.04/02 (0=авария)": DD5_DI.8, pin 24 "сброс аварий": alarmReset, pin 25 "сброс счетчика включений Н02.04/01": N0204resetCountP1, pin 26 "сброс счетчика включений Н02.04/02": N0204resetCountP2, pin 27 "сброс счетчика наработки Н02.04/01": N0204resetWorkTimeP1, pin 28 "сброс счетчика наработки Н02.04/02": N0204resetWorkTimeP2)
	(* Защита от сухого хода Н02.04 / (LS02.03) 0=сух.ход *)
	(* сброс самоподхвата реле *)
	(* Контроль открытия хотя бы одного из клапанов КЭМ *)
	(* Удержание сигнала на выключение насосов для / гарантированного сброса самоподхвата реле. *)
	(* Проверка, что фильтры 2 / ступени в регенерации (промывке) *)
	(* Проверка, что фильтры 1 / ступени в регенерации (промывке) *)
	#326 OR(pin 1, pin 2, pin 3, pin 4, pin 5, pin 6)
	#327 OR(#326, #328, #329)
	#328 OR(pin 7, pin 8, pin 9, pin 10, pin 11, pin 12)
	#329 OR(pin 13, pin 14, pin 15, pin 16)
	#330 N020401fTrigStop:F_TRIG(CLK: #337.pump1ON)
	#331 AND(#327, pin 17)
	#332 OR(#330.Q, #335.Q)
	#333 N0204stop:TOF(IN: #332, PT: T#1s)
	out 5 "стоп Н02.04" <= #333.Q
	#334 N0204chooseRegime:choosePumpRegime(start: #331, pump1Main: pin 18, pump2Main: pin 19, byCounter: #336, byWorkTime: pin 21)
	out 1 "выбран режим Н02.04/01 = главный" <= #334.pump1MainActive
	#335 N020402fTrigStop:F_TRIG(CLK: #337.pump2ON)
	out 2 "выбран режим Н02.04/02 = главный" <= #334.pump2MainActive
	out 3 "выбран режим по кол-ву включений" <= #334.byCounterActive
	#336 OR(pin 20, startInitializer)
	out 4 "выбран режим по наработке" <= #334.byWorkTimeActive
	#337 N0204manager:TwoPumpManager(startStopPump1: #334.startPump1, startStopPump2: #334.startPump2, alarmPump1: NOT pin 22, alarmPump2: NOT pin 23, alarmReset: pin 24, counterStart: #334.startByCounter, Pump1ResetCounter: pin 25, Pump2ResetCounter: pin 26, ValueToResetCounter: -, workTimeStart: #334.startByWorkTime, workTimePump1Reset: pin 27, workTimePump2Reset: pin 28)
	out 6 "пуск Н02.04/01" <= #337.pump1ON
	out 7 "пуск Н02.04/02" <= #337.pump2ON
	out 8 "счетчик включений Н02.04/01" <= #337.counterPump1
	out 9 "счетчик включений Н02.04/02" <= #337.counterPump2
	out 10 "счетчик наработки Н02.04/01" <= #337.currentWorkTimePump1
	out 11 "счетчик наработки Н02.04/02" <= #337.currentWorkTimePump2
END_MACRO
#338 N0204statRegimeP1M <= #325.out 1
#339 N0204statRegimeP2M <= #325.out 2
#340 N0204statRegimeByC <= #325.out 3
#341 N0204statRegimeWT <= #325.out 4
#342 DD4_DO.14 <= #325.out 5
#343 DD1_DO1 <= #325.out 6
#344 DD1_DO2 <= #325.out 7
#345 N0204counterP1 <= #325.out 8
#346 N0204counterP2 <= #325.out 9
#347 N0204workTimeP1 <= #325.out 10
#348 N0204workTimeP2 <= #325.out 11
#349 OR(DD6_DI.20, DD6_DI.22, DD6_DI.24, DD6_DI.26, DD6_DI.28, DD6_DI.30)
#350 OR(DD7_DI.0, DD7_DI.2, DD7_DI.4, DD7_DI.6, DD7_DI.8, DD7_DI.10)
#351 OR(DD1_DI11, DD1_DI10, DD1_DI9, DD1_DI8)
#352 OR(#349, #350, #351)
#353 AND(#352, DD5_DI.11)
#354 OR(N0204regimeByC, startInitializer)
#355 N0204chooseRegime:choosePumpRegime(start: #353, pump1Main: N0204regimeP1M, pump2Main: N0204regimeP2M, byCounter: #354, byWorkTime: N0204regimeWT)
#356 N0204statRegimeP1M <= #355.pump1MainActive
#357 N0204statRegimeP2M <= #355.pump2MainActive
#358 N0204statRegimeByC <= #355.byCounterActive
#359 N0204statRegimeWT <= #355.byWorkTimeActive
#360 N0204manager:TwoPumpManager(startStopPump1: #355.startPump1, startStopPump2: #355.startPump2, alarmPump1: NOT DD5_DI.7, alarmPump2: NOT DD5_DI.8, alarmReset: alarmReset, counterStart: #355.startByCounter, Pump1ResetCounter: N0204resetCountP1, Pump2ResetCounter: N0204resetCountP2, ValueToResetCounter: -, workTimeStart: #355.startByWorkTime, workTimePump1Reset: N0204resetWorkTimeP1, workTimePump2Reset: N0204resetWorkTimeP2)
#361 DD1_DO1 <= #360.pump1ON
#362 DD1_DO2 <= #360.pump2ON
#363 N0204counterP1 <= #360.counterPump1
#364 N0204counterP2 <= #360.counterPump2
#365 N0204workTimeP1 <= #360.currentWorkTimePump1
#366 N0204workTimeP2 <= #360.currentWorkTimePump2
#367 N020401fTrigStop:F_TRIG(CLK: #360.pump1ON)
#368 N020402fTrigStop:F_TRIG(CLK: #360.pump2ON)
#369 OR(#367.Q, #368.Q)
#370 N0204stop:TOF(IN: #369, PT: T#1s)
#371 DD4_DO.14 <= #370.Q
_END_CFC_
END_PROGRAM

(* POU DosingPumpProportional, CFC *)
FUNCTION_BLOCK DosingPumpProportional
VAR_INPUT
	flowValue: REAL;		(*текущее значение мгновенного расхода, кубометров в час.*)
	setMinPumpDosingValue: REAL := 0;		(*задание минимальной производительности доз.насоса.
По умолчанию, если ничего не подключено ко входу, равно нулю.*)
	setMaxPumpDosingValue: REAL;		(*задание максимальной производительности доз.насоса, в мл/мин*)
	minOutputValue: REAL := 4;		(*минимальное значение выходного сигнала.
По умолчанию, если ничего не подключено ко входу, равно 4.*)
	maxOutputValue: REAL := 20;		(*Максимально значение выходного сигнала.
			По умолчанию, если ничего не подключено ко входу, равно 20.*)
	setKoeffProportionality: REAL;		(*Задание мл на кубометр (коэф.пропорциональности между расходом и дозированием)*)
	minFlowToStart: REAL := 10;		(*Минимальное значение расхода для подачи сигнала на начало дозирования.
			По умолчанию, если ничего не подключено ко входу, равно 10 кубометров в час.*)
END_VAR
VAR_OUTPUT
	outputValue: REAL;		(*Выходной сигнал на дозирующий насос.*)
	dosingError: BOOL;		(*Ошибка производительности дозирования (неверно заданы значения производительности насоса, производительность доз.насоса не соответствует расходу.*)
	startDosingPump: BOOL;		(*Сигнал на запуск дозирующего насоса.*)
END_VAR
VAR
	linearTransformator: LIN_TRAFO;		(*получает на вход значение из указанного диапазона, ставит на выходе пропорциональное значение из другого диапазона.*)
END_VAR
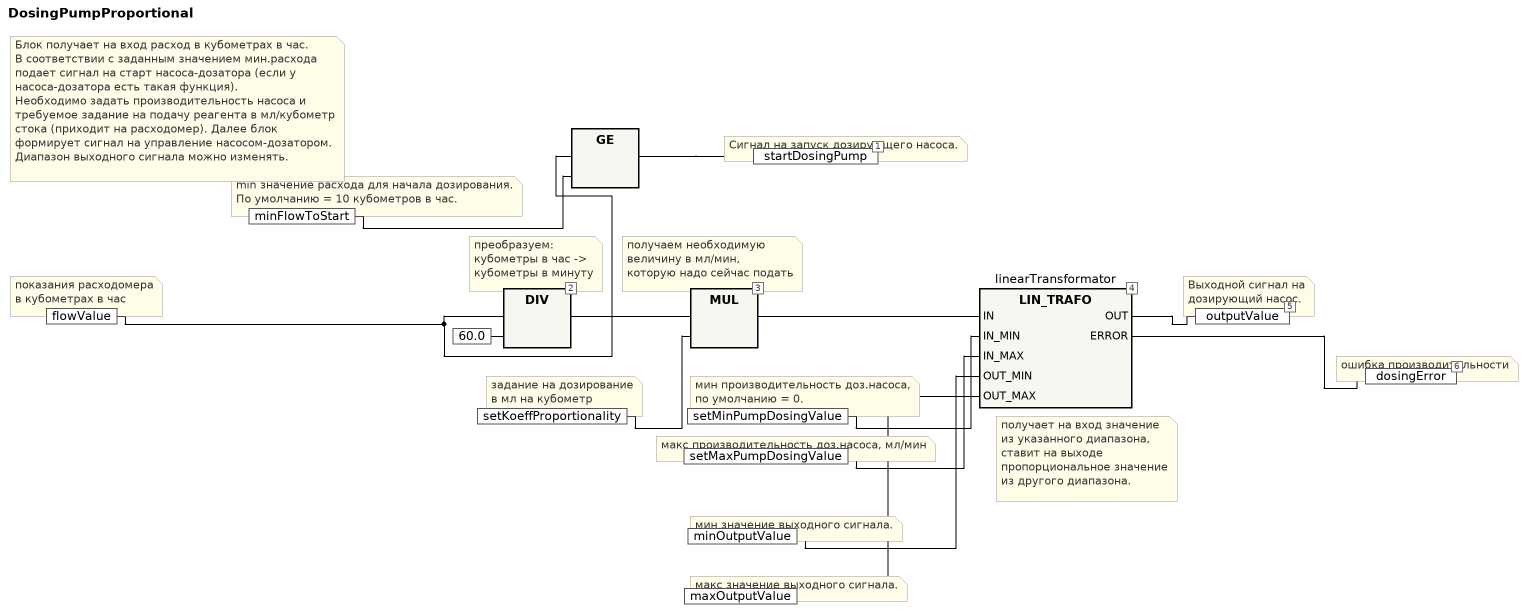
_CFC_ (* Continuous Function Chart, elements in execution order *)
(* Сигнал на запуск дозирующего насоса. *)
(* min значение расхода для начала дозирования. / По умолчанию = 10 кубометров в час. *)
(* макс производительность доз.насоса, мл/мин *)
(* мин производительность доз.насоса, / по умолчанию = 0. *)
(* получаем необходимую / величину в мл/мин, / которую надо сейчас подать *)
(* задание на дозирование / в мл на кубометр *)
(* показания расходомера / в кубометрах в час *)
(* преобразуем: / кубометры в час -> / кубометры в минуту *)
(* мин значение выходного сигнала. *)
(* макс значение выходного сигнала. *)
(* Выходной сигнал на / дозирующий насос. *)
(* ошибка производительности *)
(* получает на вход значение / из указанного диапазона, / ставит на выходе / пропорциональное значение / из другого диапазона. *)
(* Блок получает на вход расход в кубометрах в час. / В соответствии с заданным значением мин.расхода подает сигнал на старт насоса-дозатора (если у насоса-дозатора есть такая функция). / Необходимо задать производительность насоса и требуемое задание на подачу реагента в мл/кубометр стока (приходит на расходомер). Далее блок формирует сигнал на управление насосом-дозатором. / Диапазон выходного сигнала можно изменять. *)
#0 GE(flowValue, minFlowToStart)
#1 startDosingPump <= #0
#2 DIV(flowValue, 60.0)
#3 MUL(#2, setKoeffProportionality)
#4 linearTransformator:LIN_TRAFO(IN: #3, IN_MIN: setMinPumpDosingValue, IN_MAX: setMaxPumpDosingValue, OUT_MIN: minOutputValue, OUT_MAX: maxOutputValue)
#5 outputValue <= #4.OUT
#6 dosingError <= #4.ERROR
_END_CFC_
(* the same logic as Structured Text *)
(* Сигнал на запуск дозирующего насоса. *)
(* min значение расхода для начала дозирования. / По умолчанию = 10 кубометров в час. *)
(* макс производительность доз.насоса, мл/мин *)
(* мин производительность доз.насоса, / по умолчанию = 0. *)
(* получаем необходимую / величину в мл/мин, / которую надо сейчас подать *)
(* задание на дозирование / в мл на кубометр *)
(* показания расходомера / в кубометрах в час *)
(* преобразуем: / кубометры в час -> / кубометры в минуту *)
(* мин значение выходного сигнала. *)
(* макс значение выходного сигнала. *)
(* Выходной сигнал на / дозирующий насос. *)
(* ошибка производительности *)
(* получает на вход значение / из указанного диапазона, / ставит на выходе / пропорциональное значение / из другого диапазона. *)
(* Блок получает на вход расход в кубометрах в час. / В соответствии с заданным значением мин.расхода подает сигнал на старт насоса-дозатора (если у насоса-дозатора есть такая функция). / Необходимо задать производительность насоса и требуемое задание на подачу реагента в мл/кубометр стока (приходит на расходомер). Далее блок формирует сигнал на управление насосом-дозатором. / Диапазон выходного сигнала можно изменять. *)
startDosingPump := flowValue >= minFlowToStart;
linearTransformator(IN := (flowValue / 60.0) * setKoeffProportionality, IN_MIN := setMinPumpDosingValue, IN_MAX := setMaxPumpDosingValue, OUT_MIN := minOutputValue, OUT_MAX := maxOutputValue);
outputValue := linearTransformator.OUT;
dosingError := linearTransformator.ERROR;
END_FUNCTION_BLOCK

(* POU choosePumpRegime, CFC *)
FUNCTION_BLOCK choosePumpRegime
VAR
	pump1RStrig: RS;		(*Триггер-защелка выбора режима с главным первым насосом.*)
	pump2RStrig: RS;		(*Триггер-защелка выбора режима с главным вторым насосом.*)
	byCounterRStrig: RS;		(*Триггер-защелка выбора режима с запуском по количеству включений.*)
	byWorkTimeRStrig: RS;		(*Триггер-защелка выбора режима с запуском по наработке.*)
	Pump1MainDetector: R_TRIG;		(*Детектор переднего фронта включения режима, когда главный насос - первый.
			Для сброса остальных значений.*)
	Pump2MainDetector: R_TRIG;		(*Детектор переднего фронта включения режима, когда главный насос - второй.
			Для сброса остальных значений.*)
	ByCounterDetector: R_TRIG;		(*Детектор переднего фронта включения режима по количеству включений.
			Для сброса остальных значений.*)
	ByWorkTimeDetector: R_TRIG;		(*Детектор переднего фронта включения режима по наработке.
			Для сброса остальных значений.*)
END_VAR
VAR_INPUT
	start: BOOL;		(*Сигнал на включение насоса.
			Активируется выход согласно выбранного режима.*)
	pump1Main: BOOL;		(*Режим: первый насос главный, второй - резервный.*)
	pump2Main: BOOL;		(*Режим: второй насос главный, первый - резервный.*)
	byCounter: BOOL;		(*Режим: запуск по количеству включений.
			Включится с меньшим количеством стартов.*)
	byWorkTime: BOOL;		(*Режим: запуск по наработке.
			Включится насос с меньшей наработкой.*)
END_VAR
VAR_OUTPUT
	pump1MainActive: BOOL;		(*Активный режим: первый насос главный.*)
	pump2MainActive: BOOL;		(*Активный режим: второй насос главный.*)
	byCounterActive: BOOL;		(*Активный режим: включение по количеству запусков.*)
	byWorkTimeActive: BOOL;		(*Активный режим: по наработке.*)
	startPump1: BOOL;		(*Запуск первого насоса как главного (основного).*)
	startPump2: BOOL;		(*Запуск второго насоса как главного (основного).*)
	startByCounter: BOOL;		(*Запуск насоса по количеству стартов.
			Запустится с меньшим. Если одинаково, то - первый.*)
	startByWorkTime: BOOL;		(*Запуск по наработке.
			Включится с меньшей. Если одинаково, то - первый.*)
END_VAR
VAR (* helpers for the ST form of the networks *)
	_en62 : BOOL;
	_t62 : BOOL;
	_en72 : BOOL;
	_t72 : BOOL;
	_en78 : BOOL;
	_t78 : BOOL;
	_en84 : BOOL;
	_t84 : BOOL;
END_VAR
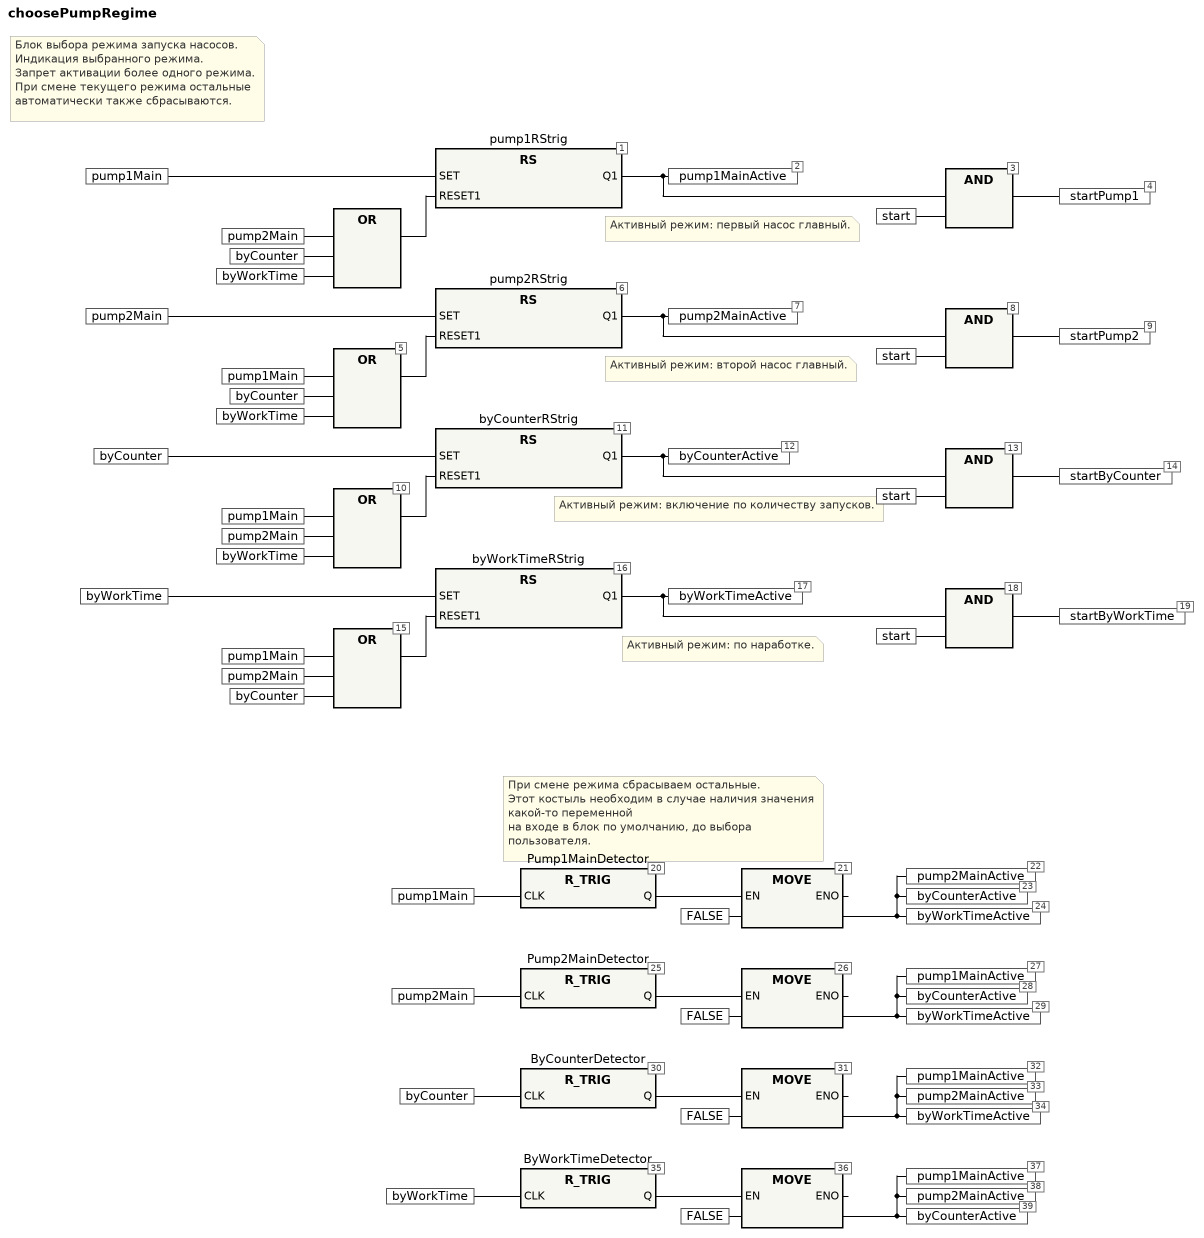
_CFC_ (* Continuous Function Chart, elements in execution order *)
(* Блок выбора режима запуска насосов. / Индикация выбранного режима. / Запрет активации более одного режима. / При смене текущего режима остальные автоматически также сбрасываются. *)
(* Активный режим: первый насос главный. *)
(* Активный режим: включение по количеству запусков. *)
(* Активный режим: по наработке. *)
(* Активный режим: второй насос главный. *)
(* При смене режима сбрасываем остальные. / Этот костыль необходим в случае наличия значения какой-то переменной / на входе в блок по умолчанию, до выбора пользователя. *)
#0 OR(pump2Main, byCounter, byWorkTime)
#1 pump1RStrig:RS(SET: pump1Main, RESET1: #0)
#2 pump1MainActive <= #1.Q1
#3 AND(#1.Q1, start)
#4 startPump1 <= #3
#5 OR(pump1Main, byCounter, byWorkTime)
#6 pump2RStrig:RS(SET: pump2Main, RESET1: #5)
#7 pump2MainActive <= #6.Q1
#8 AND(#6.Q1, start)
#9 startPump2 <= #8
#10 OR(pump1Main, pump2Main, byWorkTime)
#11 byCounterRStrig:RS(SET: byCounter, RESET1: #10)
#12 byCounterActive <= #11.Q1
#13 AND(#11.Q1, start)
#14 startByCounter <= #13
#15 OR(pump1Main, pump2Main, byCounter)
#16 byWorkTimeRStrig:RS(SET: byWorkTime, RESET1: #15)
#17 byWorkTimeActive <= #16.Q1
#18 AND(#16.Q1, start)
#19 startByWorkTime <= #18
#20 Pump1MainDetector:R_TRIG(CLK: pump1Main)
#21 MOVE(EN: #20.Q, FALSE)
#22 pump2MainActive <= #21
#23 byCounterActive <= #21
#24 byWorkTimeActive <= #21
#25 Pump2MainDetector:R_TRIG(CLK: pump2Main)
#26 MOVE(EN: #25.Q, FALSE)
#27 pump1MainActive <= #26
#28 byCounterActive <= #26
#29 byWorkTimeActive <= #26
#30 ByCounterDetector:R_TRIG(CLK: byCounter)
#31 MOVE(EN: #30.Q, FALSE)
#32 pump1MainActive <= #31
#33 pump2MainActive <= #31
#34 byWorkTimeActive <= #31
#35 ByWorkTimeDetector:R_TRIG(CLK: byWorkTime)
#36 MOVE(EN: #35.Q, FALSE)
#37 pump1MainActive <= #36
#38 pump2MainActive <= #36
#39 byCounterActive <= #36
_END_CFC_
(* the same logic as Structured Text *)
(* Блок выбора режима запуска насосов. / Индикация выбранного режима. / Запрет активации более одного режима. / При смене текущего режима остальные автоматически также сбрасываются. *)
(* Активный режим: первый насос главный. *)
(* Активный режим: включение по количеству запусков. *)
(* Активный режим: по наработке. *)
(* Активный режим: второй насос главный. *)
(* При смене режима сбрасываем остальные. / Этот костыль необходим в случае наличия значения какой-то переменной / на входе в блок по умолчанию, до выбора пользователя. *)
pump1RStrig(SET := pump1Main, RESET1 := pump2Main OR byCounter OR byWorkTime);
pump1MainActive := pump1RStrig.Q1;
startPump1 := pump1RStrig.Q1 AND start;
pump2RStrig(SET := pump2Main, RESET1 := pump1Main OR byCounter OR byWorkTime);
pump2MainActive := pump2RStrig.Q1;
startPump2 := pump2RStrig.Q1 AND start;
byCounterRStrig(SET := byCounter, RESET1 := pump1Main OR pump2Main OR byWorkTime);
byCounterActive := byCounterRStrig.Q1;
startByCounter := byCounterRStrig.Q1 AND start;
byWorkTimeRStrig(SET := byWorkTime, RESET1 := pump1Main OR pump2Main OR byCounter);
byWorkTimeActive := byWorkTimeRStrig.Q1;
startByWorkTime := byWorkTimeRStrig.Q1 AND start;
Pump1MainDetector(CLK := pump1Main);
_en62 := Pump1MainDetector.Q;
IF _en62 THEN _t62 := FALSE; END_IF;
IF _en62 THEN pump2MainActive := _t62; END_IF;
IF _en62 THEN byCounterActive := _t62; END_IF;
IF _en62 THEN byWorkTimeActive := _t62; END_IF;
Pump2MainDetector(CLK := pump2Main);
_en72 := Pump2MainDetector.Q;
IF _en72 THEN _t72 := FALSE; END_IF;
IF _en72 THEN pump1MainActive := _t72; END_IF;
IF _en72 THEN byCounterActive := _t72; END_IF;
IF _en72 THEN byWorkTimeActive := _t72; END_IF;
ByCounterDetector(CLK := byCounter);
_en78 := ByCounterDetector.Q;
IF _en78 THEN _t78 := FALSE; END_IF;
IF _en78 THEN pump1MainActive := _t78; END_IF;
IF _en78 THEN pump2MainActive := _t78; END_IF;
IF _en78 THEN byWorkTimeActive := _t78; END_IF;
ByWorkTimeDetector(CLK := byWorkTime);
_en84 := ByWorkTimeDetector.Q;
IF _en84 THEN _t84 := FALSE; END_IF;
IF _en84 THEN pump1MainActive := _t84; END_IF;
IF _en84 THEN pump2MainActive := _t84; END_IF;
IF _en84 THEN byCounterActive := _t84; END_IF;
END_FUNCTION_BLOCK

(* POU TwoPumpManager, CFC *)
FUNCTION_BLOCK TwoPumpManager
VAR_INPUT
	startStopPump1: BOOL;		(*Сигнал на пуск/стоп первого насоса.*)
	startStopPump2: BOOL;		(*Сигнал на пуск/стоп второго насоса.*)
	alarmPump1: BOOL;		(*Сигнал "авария" на первом насосе.*)
	alarmPump2: BOOL;		(*Сигнал "авария" на втором насосе.*)
	alarmReset: BOOL;		(*Сброс аварии.*)

	counterStart: BOOL;		(*Запуск насоса с меньшим количеством включений.*)
	Pump1ResetCounter: BOOL;		(*Сброс счетчика количества включений первого насоса.
Сбрасывается также автоматически при достижении счетчиком значения ValueToResetCTU.*)
	Pump2ResetCounter: BOOL;		(*Сброс счетчика количества включений второго насоса.
Сбрасывается также автоматически при достижении счетчиком значения ValueToResetCTU.*)
	ValueToResetCounter: WORD := 32767;		(*Значение счетчика, после которого он сбрасывается на ноль.
			Максимальное допустимое значение: 32767, будет установлено, если не подключать ничего на вход.*)

	workTimeStart: BOOL;		(*Запуск насоса с выбором по меньшей наработке.*)
	workTimePump1Reset: BOOL;		(*Сброс времени наработки первого насоса.*)
	workTimePump2Reset: BOOL;		(*Сброс времени наработки второго насоса.*)
END_VAR
VAR_OUTPUT
	pump1ON: BOOL;		(*Выход на включение первого насоса.*)
	pump2ON: BOOL;		(*Выход на включение второго насоса.*)

	counterPump1: WORD;		(*Количество включений первого насоса.
При достижении значения ValueToResetCTU сбрасывается в ноль.*)
	counterPump2: WORD;		(*Количество включений второго насоса.
При достижении значения ValueToResetCTU сбрасывается в ноль.*)

	currentWorkTimePump1: TIME;		(*Текущая наработка первого насоса.*)
	currentWorkTimePump2: TIME;		(*Текущая наработка второго насоса.*)
END_VAR
VAR
	RtrigPump1: R_TRIG;		(*Включает первый насос по фронту сигнала на ручной пуск/стоп.*)
	FtrigPump1: F_TRIG;		(*Выключает первый насос по спаду сигнала на ручной пуск/стоп.*)
	RtrigPump2: R_TRIG;		(*Включает второй насос по фронту сигнала на ручной пуск/стоп.*)
	FtrigPump2: F_TRIG;		(*Выключает второй насос по спаду сигнала на ручной пуск/стоп.*)
	RSpump1: RS;		(*RS-триггер нормального включения первого насоса*)
	RSpump2: RS;		(*RS-триггер нормального включения второго насоса*)
	pump1NormalON: BOOL;		(*Сигнал нормального (неаварийного) включения первого насоса.*)
	pump2NormalON: BOOL;		(*Сигнал нормального (неаварийного) включения второго насоса.*)
	pump2EmergencyON: BOOL;		(*Сигнал аварийного включения второго насоса (при аварии первого).*)
	pump1EmergencyON: BOOL;		(*Сигнал аварийного включения первого насоса (при аварии второго).*)
	alarmPump1RStrig: RS;		(*Триггер аварии первого насоса.*)
	alarmPump2RStrig: RS;		(*Триггер аварии второго насоса.*)
	TONtoOnPump1: TON;		(*Таймер задержки включения первого насоса, на переключение контакторов при аварийном переключении.
			Жестко задано 1 секунда.*)
	TONtoOnPump2: TON;		(*Таймер задержки включения второго насоса, на переключение контакторов при аварийном переключении.
						Жестко задано 1 секунда.*)

	CTUPump1: CTU;		(*Счетчик количества включений первого насоса.*)
	CTUPump2: CTU;		(*Счетчик количества включений второго насоса.*)
	counterRtrig: R_TRIG;		(*Детектор переднего фронта сигнала на старт насоса с меньшей наработкой, включает насос.*)
	counterFtrig: F_TRIG;		(*Детектор спада сигнала на запуск насоса с меньшей наработкой, останавливает насос.*)
	counterRStrigPump1: RS;		(*Триггер-защелка включения первого насоса при запуске по количеству включений.*)
	counterRStrigPump2: RS;		(*Триггер-защелка включения второго насоса при запуске по количеству включений.*)
	counterPump1ON: BOOL;		(*Сигнал на запуск первого насоса при запуске по количеству включений.*)
	counterPump2ON: BOOL;		(*Сигнал на запуск второго насоса при запуске по количеству включений.*)

	workTimePump1ON: BOOL;		(*Сигнал на запуск первого насоса при запуске по наработке.*)
	workTimePump2ON: BOOL;		(*Сигнал на запуск второго насоса при запуске по наработке.*)
	timerFtrig: F_TRIG;		(*Детектор спада сигнала работы насосов для записи времени работы.*)
	pump1Ftrig: F_TRIG;		(*Детектор спада сигнала работы первого насоса для подсчета наработки.*)
	pump2Ftrig: F_TRIG;		(*Детектор спада сигнала работы второго насоса для подсчета наработки.*)
	timeStartFtrig: F_TRIG;		(*Детектор спада сигнала на запуск по наработке.*)
	timeStartRtrig: R_TRIG;		(*Детектор переднего фронта сигнала на запуск по наработке.*)
	timerRTC: RTC;		(*Таймер реального времени для подсчета наработки.*)
	timeCDT: DT;		(*Время на выходе таймера реального времени.*)
	timePDT: DT;		(*Время на входе таймера реального времени. Не инициализируется, чтобы подсчет всегда начинался от нуля.*)
	tempVarTime: TIME;		(*Промежуточная переменная хранения времени наработки за включение.*)
	workTimePump1: TIME;		(*Время наработки первого насоса. Подсчитывается после выключения насоса.*)
	workTimePump2: TIME;		(*Время наработки второго насоса. Подсчитывается после выключения насоса.*)
	RStrigTimePump1: RS;		(*Триггер-защелка запуск первого насоса по наработке.*)
	RStrigTimePump2: RS;		(*Триггер-защелка запуск второго насоса по наработке.*)

END_VAR
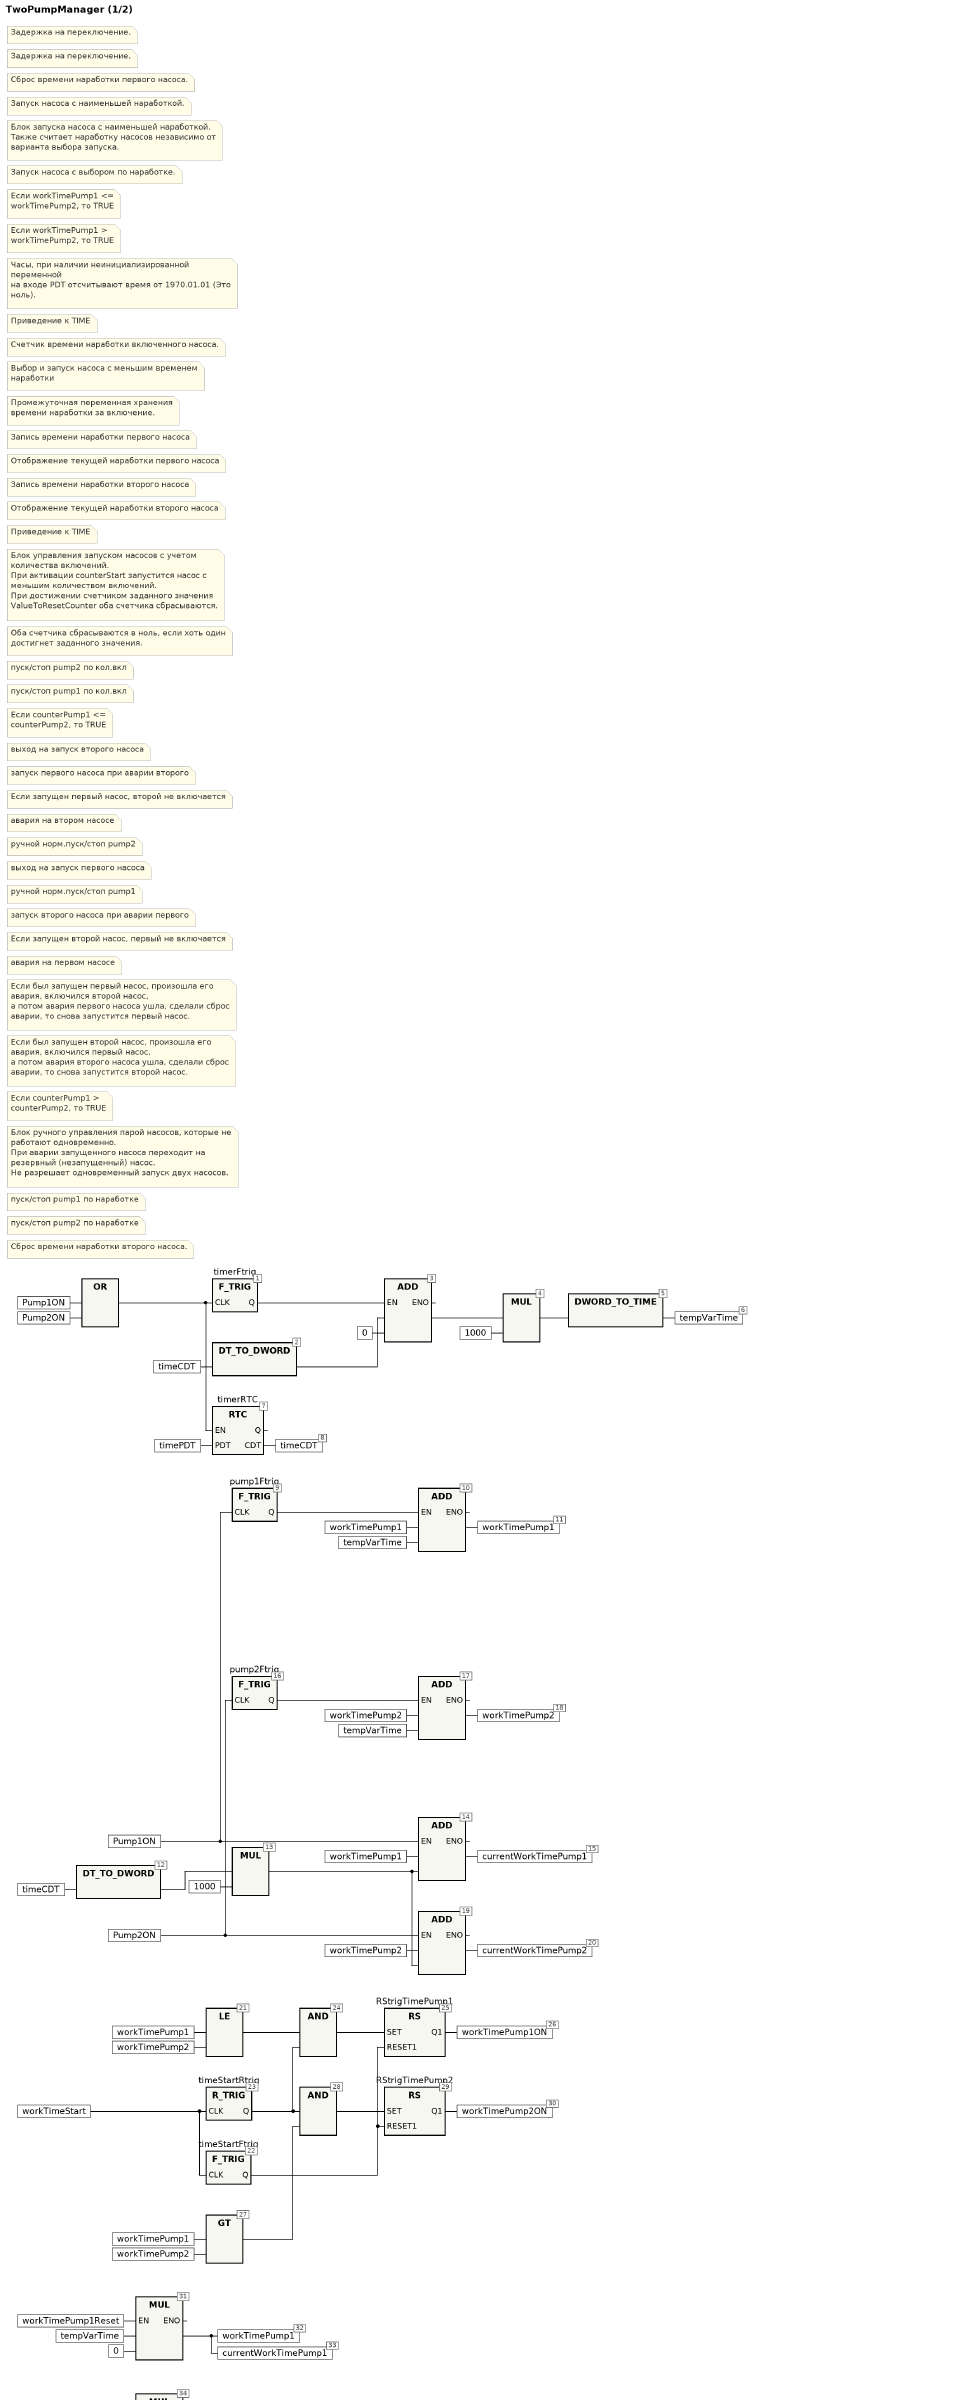
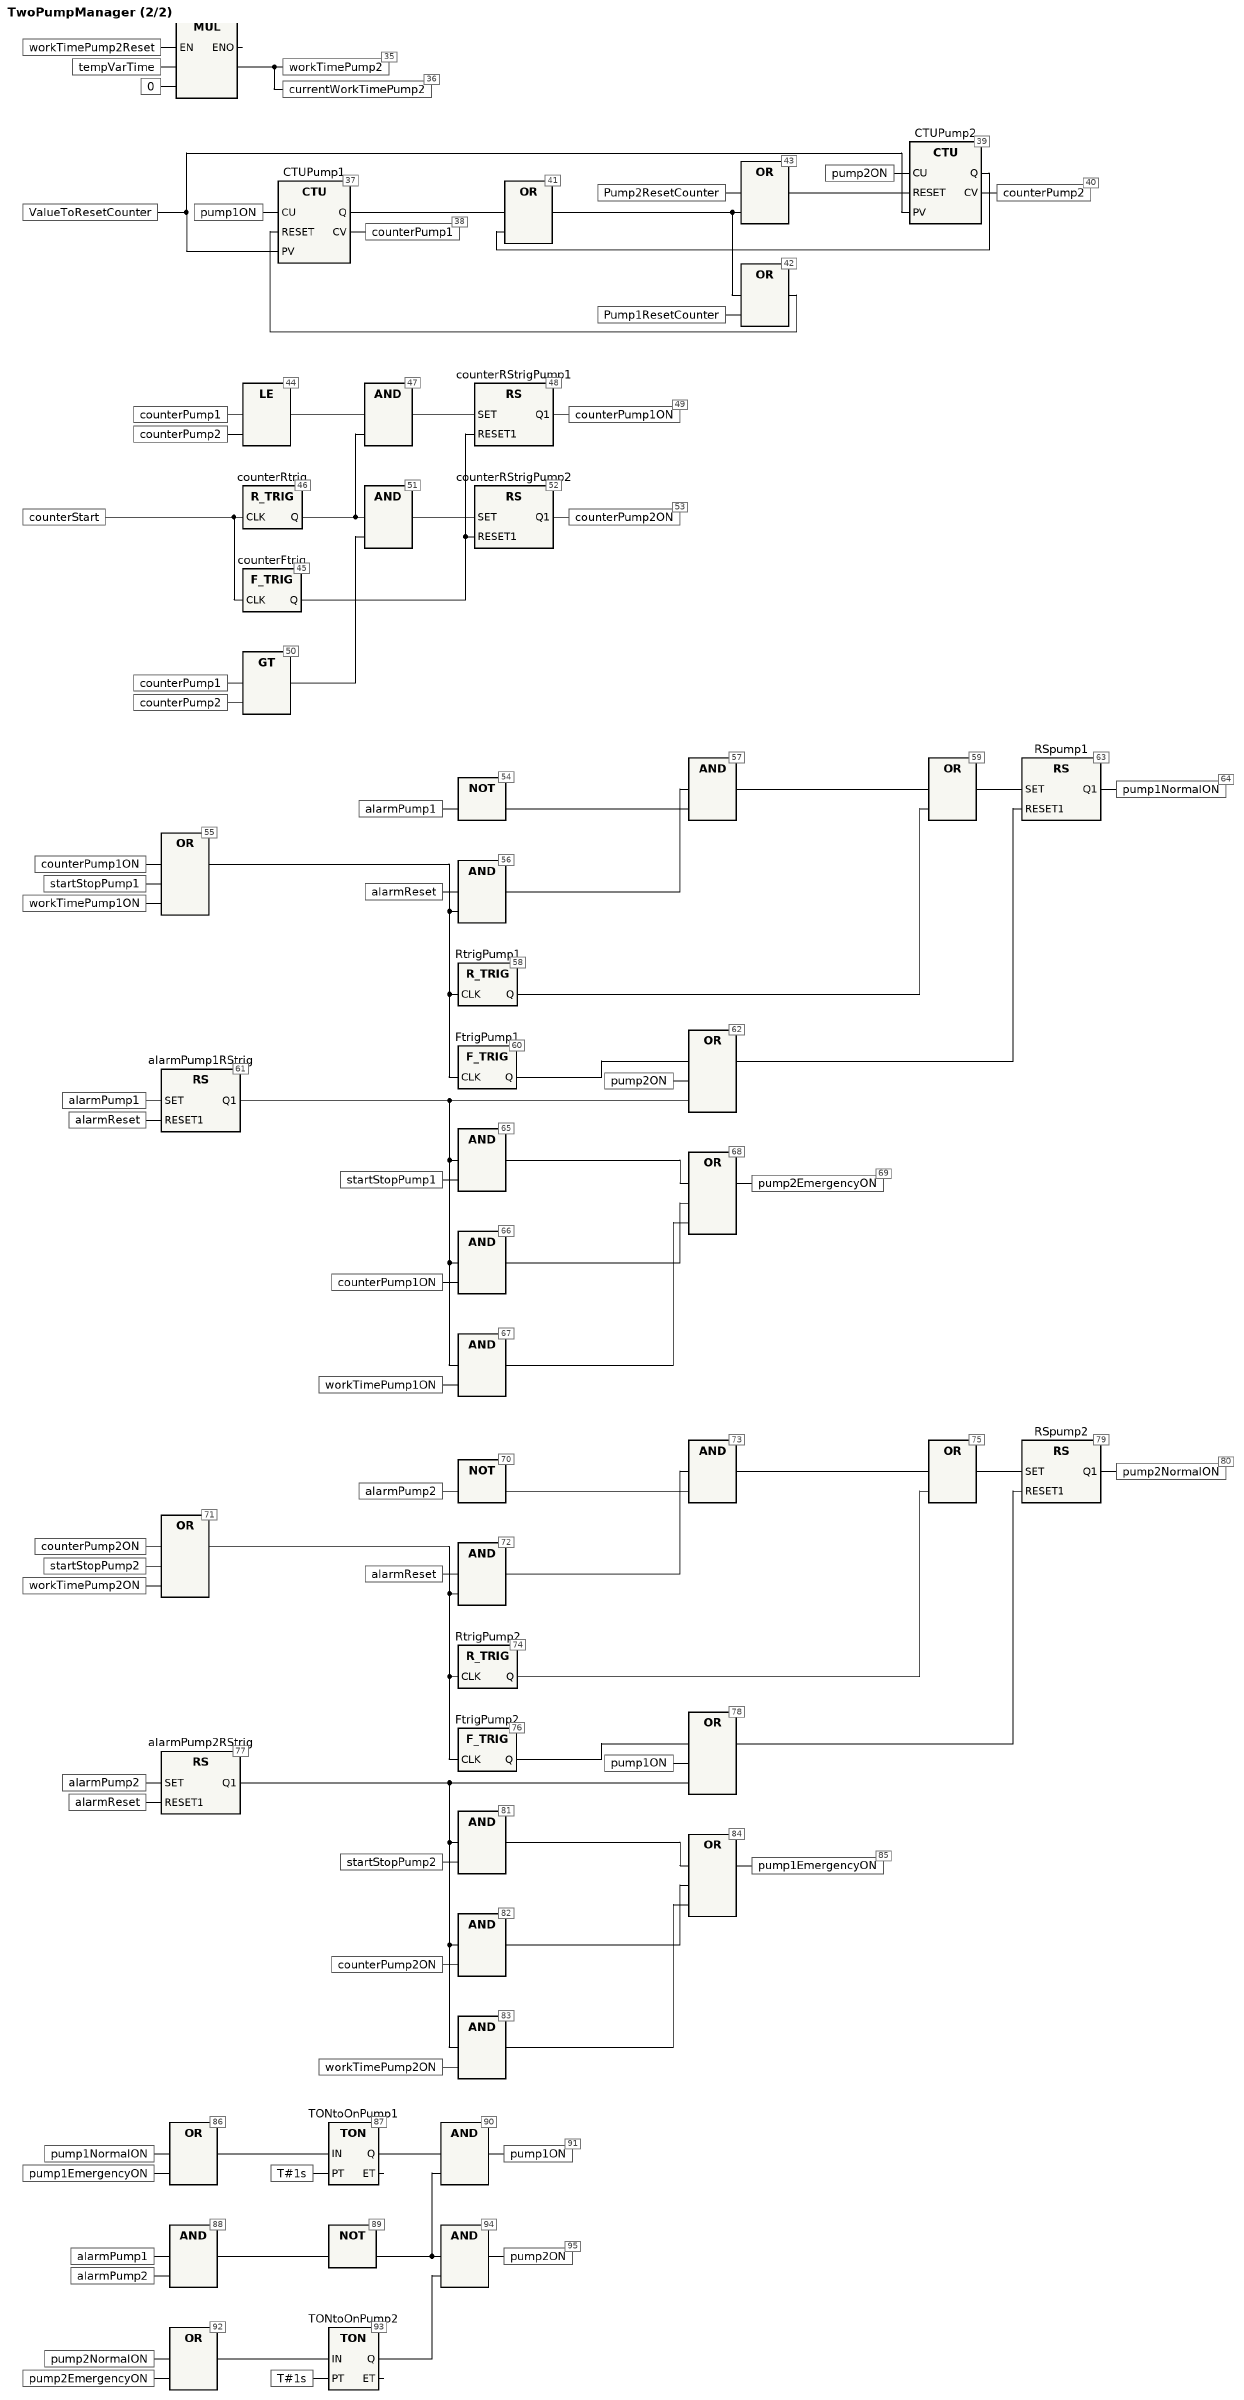
_CFC_ (* Continuous Function Chart, elements in execution order *)
(* Задержка на переключение. *)
(* Задержка на переключение. *)
(* Сброс времени наработки первого насоса. *)
(* Запуск насоса с наименьшей наработкой. *)
(* Блок запуска насоса с наименьшей наработкой. / Также считает наработку насосов независимо от варианта выбора запуска. *)
(* Запуск насоса с выбором по наработке. *)
(* Если workTimePump1 <= / workTimePump2, то TRUE *)
(* Если workTimePump1 > / workTimePump2, то TRUE *)
(* Часы, при наличии неинициализированной переменной / на входе PDT отсчитывают время от 1970.01.01 (Это ноль). *)
(* Приведение к TIME *)
(* Счетчик времени наработки включенного насоса. *)
(* Выбор и запуск насоса с меньшим временем наработки *)
(* Промежуточная переменная хранения / времени наработки за включение. *)
(* Запись времени наработки первого насоса *)
(* Отображение текущей наработки первого насоса *)
(* Запись времени наработки второго насоса *)
(* Отображение текущей наработки второго насоса *)
(* Приведение к TIME *)
(* Блок управления запуском насосов с учетом количества включений. / При активации counterStart запустится насос с меньшим количеством включений. / При достижении счетчиком заданного значения ValueToResetCounter оба счетчика сбрасываются. *)
(* Оба счетчика сбрасываются в ноль, если хоть один достигнет заданного значения. *)
(* пуск/стоп pump2 по кол.вкл *)
(* пуск/стоп pump1 по кол.вкл *)
(* Если counterPump1 <= / counterPump2, то TRUE *)
(* выход на запуск второго насоса *)
(* запуск первого насоса при аварии второго *)
(* Если запущен первый насос, второй не включается *)
(* авария на втором насосе *)
(* ручной норм.пуск/стоп pump2 *)
(* выход на запуск первого насоса *)
(* ручной норм.пуск/стоп pump1 *)
(* запуск второго насоса при аварии первого *)
(* Если запущен второй насос, первый не включается *)
(* авария на первом насосе *)
(* Если был запущен первый насос, произошла его авария, включился второй насос, / а потом авария первого насоса ушла, сделали сброс аварии, то снова запустится первый насос. *)
(* Если был запущен второй насос, произошла его авария, включился первый насос, / а потом авария второго насоса ушла, сделали сброс аварии, то снова запустится второй насос. *)
(* Если counterPump1 > / counterPump2, то TRUE *)
(* Блок ручного управления парой насосов, которые не работают одновременно. / При аварии запущенного насоса переходит на резервный (незапущенный) насос. / Не разрешает одновременный запуск двух насосов. *)
(* пуск/стоп pump1 по наработке *)
(* пуск/стоп pump2 по наработке *)
(* Сброс времени наработки второго насоса. *)
#0 OR(Pump1ON, Pump2ON)
#1 timerFtrig:F_TRIG(CLK: #0)
#2 DT_TO_DWORD(timeCDT)
#3 ADD(EN: #1.Q, #2, 0)
#4 MUL(#3, 1000)
#5 DWORD_TO_TIME(#4)
#6 tempVarTime <= #5
#7 timerRTC:RTC(EN: #0, PDT: timePDT)
#8 timeCDT <= #7.CDT
#9 pump1Ftrig:F_TRIG(CLK: Pump1ON)
#10 ADD(EN: #9.Q, workTimePump1, tempVarTime)
#11 workTimePump1 <= #10
#12 DT_TO_DWORD(timeCDT)
#13 MUL(#12, 1000)
#14 ADD(EN: Pump1ON, workTimePump1, #13)
#15 currentWorkTimePump1 <= #14
#16 pump2Ftrig:F_TRIG(CLK: Pump2ON)
#17 ADD(EN: #16.Q, workTimePump2, tempVarTime)
#18 workTimePump2 <= #17
#19 ADD(EN: Pump2ON, workTimePump2, #13)
#20 currentWorkTimePump2 <= #19
#21 LE(workTimePump1, workTimePump2)
#22 timeStartFtrig:F_TRIG(CLK: workTimeStart)
#23 timeStartRtrig:R_TRIG(CLK: workTimeStart)
#24 AND(#21, #23.Q)
#25 RStrigTimePump1:RS(SET: #24, RESET1: #22.Q)
#26 workTimePump1ON <= #25.Q1
#27 GT(workTimePump1, workTimePump2)
#28 AND(#23.Q, #27)
#29 RStrigTimePump2:RS(SET: #28, RESET1: #22.Q)
#30 workTimePump2ON <= #29.Q1
#31 MUL(EN: workTimePump1Reset, tempVarTime, 0)
#32 workTimePump1 <= #31
#33 currentWorkTimePump1 <= #31
#34 MUL(EN: workTimePump2Reset, tempVarTime, 0)
#35 workTimePump2 <= #34
#36 currentWorkTimePump2 <= #34
#37 CTUPump1:CTU(CU: pump1ON, RESET: #42, PV: ValueToResetCounter)
#38 counterPump1 <= #37.CV
#39 CTUPump2:CTU(CU: pump2ON, RESET: #43, PV: ValueToResetCounter)
#40 counterPump2 <= #39.CV
#41 OR(#37.Q, #39.Q)
#42 OR(#41, Pump1ResetCounter)
#43 OR(Pump2ResetCounter, #41)
#44 LE(counterPump1, counterPump2)
#45 counterFtrig:F_TRIG(CLK: counterStart)
#46 counterRtrig:R_TRIG(CLK: counterStart)
#47 AND(#44, #46.Q)
#48 counterRStrigPump1:RS(SET: #47, RESET1: #45.Q)
#49 counterPump1ON <= #48.Q1
#50 GT(counterPump1, counterPump2)
#51 AND(#46.Q, #50)
#52 counterRStrigPump2:RS(SET: #51, RESET1: #45.Q)
#53 counterPump2ON <= #52.Q1
#54 NOT(alarmPump1)
#55 OR(counterPump1ON, startStopPump1, workTimePump1ON)
#56 AND(alarmReset, #55)
#57 AND(#56, #54)
#58 RtrigPump1:R_TRIG(CLK: #55)
#59 OR(#57, #58.Q)
#60 FtrigPump1:F_TRIG(CLK: #55)
#61 alarmPump1RStrig:RS(SET: alarmPump1, RESET1: alarmReset)
#62 OR(#60.Q, pump2ON, #61.Q1)
#63 RSpump1:RS(SET: #59, RESET1: #62)
#64 pump1NormalON <= #63.Q1
#65 AND(#61.Q1, startStopPump1)
#66 AND(#61.Q1, counterPump1ON)
#67 AND(#61.Q1, workTimePump1ON)
#68 OR(#65, #66, #67)
#69 pump2EmergencyON <= #68
#70 NOT(alarmPump2)
#71 OR(counterPump2ON, startStopPump2, workTimePump2ON)
#72 AND(alarmReset, #71)
#73 AND(#72, #70)
#74 RtrigPump2:R_TRIG(CLK: #71)
#75 OR(#73, #74.Q)
#76 FtrigPump2:F_TRIG(CLK: #71)
#77 alarmPump2RStrig:RS(SET: alarmPump2, RESET1: alarmReset)
#78 OR(#76.Q, pump1ON, #77.Q1)
#79 RSpump2:RS(SET: #75, RESET1: #78)
#80 pump2NormalON <= #79.Q1
#81 AND(#77.Q1, startStopPump2)
#82 AND(#77.Q1, counterPump2ON)
#83 AND(#77.Q1, workTimePump2ON)
#84 OR(#81, #82, #83)
#85 pump1EmergencyON <= #84
#86 OR(pump1NormalON, pump1EmergencyON)
#87 TONtoOnPump1:TON(IN: #86, PT: T#1s)
#88 AND(alarmPump1, alarmPump2)
#89 NOT(#88)
#90 AND(#87.Q, #89)
#91 pump1ON <= #90
#92 OR(pump2NormalON, pump2EmergencyON)
#93 TONtoOnPump2:TON(IN: #92, PT: T#1s)
#94 AND(#89, #93.Q)
#95 pump2ON <= #94
_END_CFC_
END_FUNCTION_BLOCK

(* POU TwoPumpOneDriveManager, CFC *)
FUNCTION_BLOCK TwoPumpOneDriveManager
VAR_INPUT
	startStopPump1: BOOL;		(*Сигнал на пуск/стоп первого насоса.*)
	startStopPump2: BOOL;		(*Сигнал на пуск/стоп второго насоса.*)
	alarmPump1: BOOL;		(*Сигнал "авария" на первом насосе.*)
	alarmPump2: BOOL;		(*Сигнал "авария" на втором насосе.*)
	alarmReset: BOOL;		(*Сброс аварии.*)

	counterStart: BOOL;		(*Запуск насоса с меньшим количеством включений.*)
	Pump1ResetCounter: BOOL;		(*Сброс счетчика количества включений первого насоса.
Сбрасывается также автоматически при достижении счетчиком значения ValueToResetCTU.*)
	Pump2ResetCounter: BOOL;		(*Сброс счетчика количества включений второго насоса.
Сбрасывается также автоматически при достижении счетчиком значения ValueToResetCTU.*)
	ValueToResetCounter: WORD := 32767;		(*Значение счетчика, после которого он сбрасывается на ноль.
			Максимальное допустимое значение: 32767, будет установлено, если не подключать ничего на вход.*)

	workTimeStart: BOOL;		(*Запуск насоса с выбором по меньшей наработке.*)
	workTimePump1Reset: BOOL;		(*Сброс времени наработки первого насоса.*)
	workTimePump2Reset: BOOL;		(*Сброс времени наработки второго насоса.*)
	timeKM1off: TIME := T#20s;		(*Время на которое отключается питание ЧРП.
			По умолчанию = 20сек.*)
	timeKM23DelayON: TIME := T#15s;		(*Время задержки включения контактора насоса.
			По умолчанию = 15 сек.*)
	timeKM23offDelay: TIME := T#10s;		(*Время задержки выключения контактора насосов.
			По умолчанию = 10сек. (Чтобы сначала отключилось питание ЧРП).*)
	timeReadyToStartDelay: TIME := T#5s;		(*Время задержки подачи сигнала на старт ЧРП.
			По умолчанию = 5сек.*)
END_VAR
VAR_OUTPUT

	counterPump1: WORD;		(*Количество включений первого насоса.
При достижении значения ValueToResetCTU сбрасывается в ноль.*)
	counterPump2: WORD;		(*Количество включений второго насоса.
При достижении значения ValueToResetCTU сбрасывается в ноль.*)

	currentWorkTimePump1: TIME;		(*Текущая наработка первого насоса.*)
	currentWorkTimePump2: TIME;		(*Текущая наработка второго насоса.*)

	DriveKM: BOOL;		(*Выход на включение контактора частотного преобразователя (питание).*)
	pump1KM: BOOL;		(*Выход на включение контактора первого насоса.*)
	pump2KM: BOOL;		(*Выход на включение контактора второго насоса.*)
	driveStart: BOOL;		(*Сигнал на старт частотного преобразователя.*)
	pump1active: BOOL;		(*Идет процесс запуска насоса 1.*)
	pump2active: BOOL;		(*Идет процесс запуска насоса 2.*)
END_VAR
VAR
	RtrigPump1: R_TRIG;		(*Включает первый насос по фронту сигнала на ручной пуск/стоп.*)
	FtrigPump1: F_TRIG;		(*Выключает первый насос по спаду сигнала на ручной пуск/стоп.*)
	RtrigPump2: R_TRIG;		(*Включает второй насос по фронту сигнала на ручной пуск/стоп.*)
	FtrigPump2: F_TRIG;		(*Выключает второй насос по спаду сигнала на ручной пуск/стоп.*)
	RSpump1: RS;		(*RS-триггер нормального включения первого насоса*)
	RSpump2: RS;		(*RS-триггер нормального включения второго насоса*)
	pump1NormalON: BOOL;		(*Сигнал нормального (неаварийного) включения первого насоса.*)
	pump2NormalON: BOOL;		(*Сигнал нормального (неаварийного) включения второго насоса.*)
	pump2EmergencyON: BOOL;		(*Сигнал аварийного включения второго насоса (при аварии первого).*)
	pump1EmergencyON: BOOL;		(*Сигнал аварийного включения первого насоса (при аварии второго).*)
	alarmPump1RStrig: RS;		(*Триггер аварии первого насоса.*)
	alarmPump2RStrig: RS;		(*Триггер аварии второго насоса.*)
	TONtoOnPump1: TON;		(*Таймер задержки включения первого насоса, на переключение контакторов при аварийном переключении.
			Жестко задано 1 секунда.*)
	TONtoOnPump2: TON;		(*Таймер задержки включения второго насоса, на переключение контакторов при аварийном переключении.
						Жестко задано 1 секунда.*)

	CTUPump1: CTU;		(*Счетчик количества включений первого насоса.*)
	CTUPump2: CTU;		(*Счетчик количества включений второго насоса.*)
	counterRtrig: R_TRIG;		(*Детектор переднего фронта сигнала на старт насоса с меньшей наработкой, включает насос.*)
	counterFtrig: F_TRIG;		(*Детектор спада сигнала на запуск насоса с меньшей наработкой, останавливает насос.*)
	counterRStrigPump1: RS;		(*Триггер-защелка включения первого насоса при запуске по количеству включений.*)
	counterRStrigPump2: RS;		(*Триггер-защелка включения второго насоса при запуске по количеству включений.*)
	counterPump1ON: BOOL;		(*Сигнал на запуск первого насоса при запуске по количеству включений.*)
	counterPump2ON: BOOL;		(*Сигнал на запуск второго насоса при запуске по количеству включений.*)

	workTimePump1ON: BOOL;		(*Сигнал на запуск первого насоса при запуске по наработке.*)
	workTimePump2ON: BOOL;		(*Сигнал на запуск второго насоса при запуске по наработке.*)
	timerFtrig: F_TRIG;		(*Детектор спада сигнала работы насосов для записи времени работы.*)
	pump1Ftrig: F_TRIG;		(*Детектор спада сигнала работы первого насоса для подсчета наработки.*)
	pump2Ftrig: F_TRIG;		(*Детектор спада сигнала работы второго насоса для подсчета наработки.*)
	timeStartFtrig: F_TRIG;		(*Детектор спада сигнала на запуск по наработке.*)
	timeStartRtrig: R_TRIG;		(*Детектор переднего фронта сигнала на запуск по наработке.*)
	timerRTC: RTC;		(*Таймер реального времени для подсчета наработки.*)
	timeCDT: DT;		(*Время на выходе таймера реального времени.*)
	timePDT: DT;		(*Время на входе таймера реального времени. Не инициализируется, чтобы подсчет всегда начинался от нуля.*)
	tempVarTime: TIME;		(*Промежуточная переменная хранения времени наработки за включение.*)
	workTimePump1: TIME;		(*Время наработки первого насоса. Подсчитывается после выключения насоса.*)
	workTimePump2: TIME;		(*Время наработки второго насоса. Подсчитывается после выключения насоса.*)
	RStrigTimePump1: RS;		(*Триггер-защелка запуск первого насоса по наработке.*)
	RStrigTimePump2: RS;		(*Триггер-защелка запуск второго насоса по наработке.*)

	pump1ON: BOOL;		(*Выход на включение первого насоса.*)
	pump2ON: BOOL;		(*Выход на включение второго насоса.*)
	rTrigPump1ON: R_TRIG;		(*Детектор переднего фронта на запуск насоса 1.*)
	rTrigPump2ON: R_TRIG;		(*Детектор переднего фрона на запуск насоса 2.*)
	rTrigKM1off: R_TRIG;		(*Детектор переднего фронта сигнала на запуск одного из насосов,
			для выключения контактора КМ1 питающего ЧРП.*)
	rsTrigKM1: RS;		(*Триггер управления КМ1 (питание ЧРП).*)
	rsTrigKMpump1: RS;		(*Триггер контактора насоса 1.*)
	rsTrigKMpump2: RS;		(*Триггер контактора насоса 2.*)
	timerKM1off: TOF;		(*Таймер выключения контактора питания ЧРП.*)
	timerKM2DelayON: TON;		(*Таймер задержки включения контактора насоса 1.*)
	timerKM3DelayON: TON;		(*Таймер задержки включения контактора насоса 2.*)
	timerKM2DelayOFF: TOF;		(*Таймер задержки выключения контактора насоса 1.*)
	timerKM3DelayOFF: TOF;		(*Таймер задержки выключения контактора насоса 2.*)
	timerReadyToStartON: TON;		(*Таймер задержки подачи сигнала о готовности к старту (запуск ЧРП).*)
END_VAR
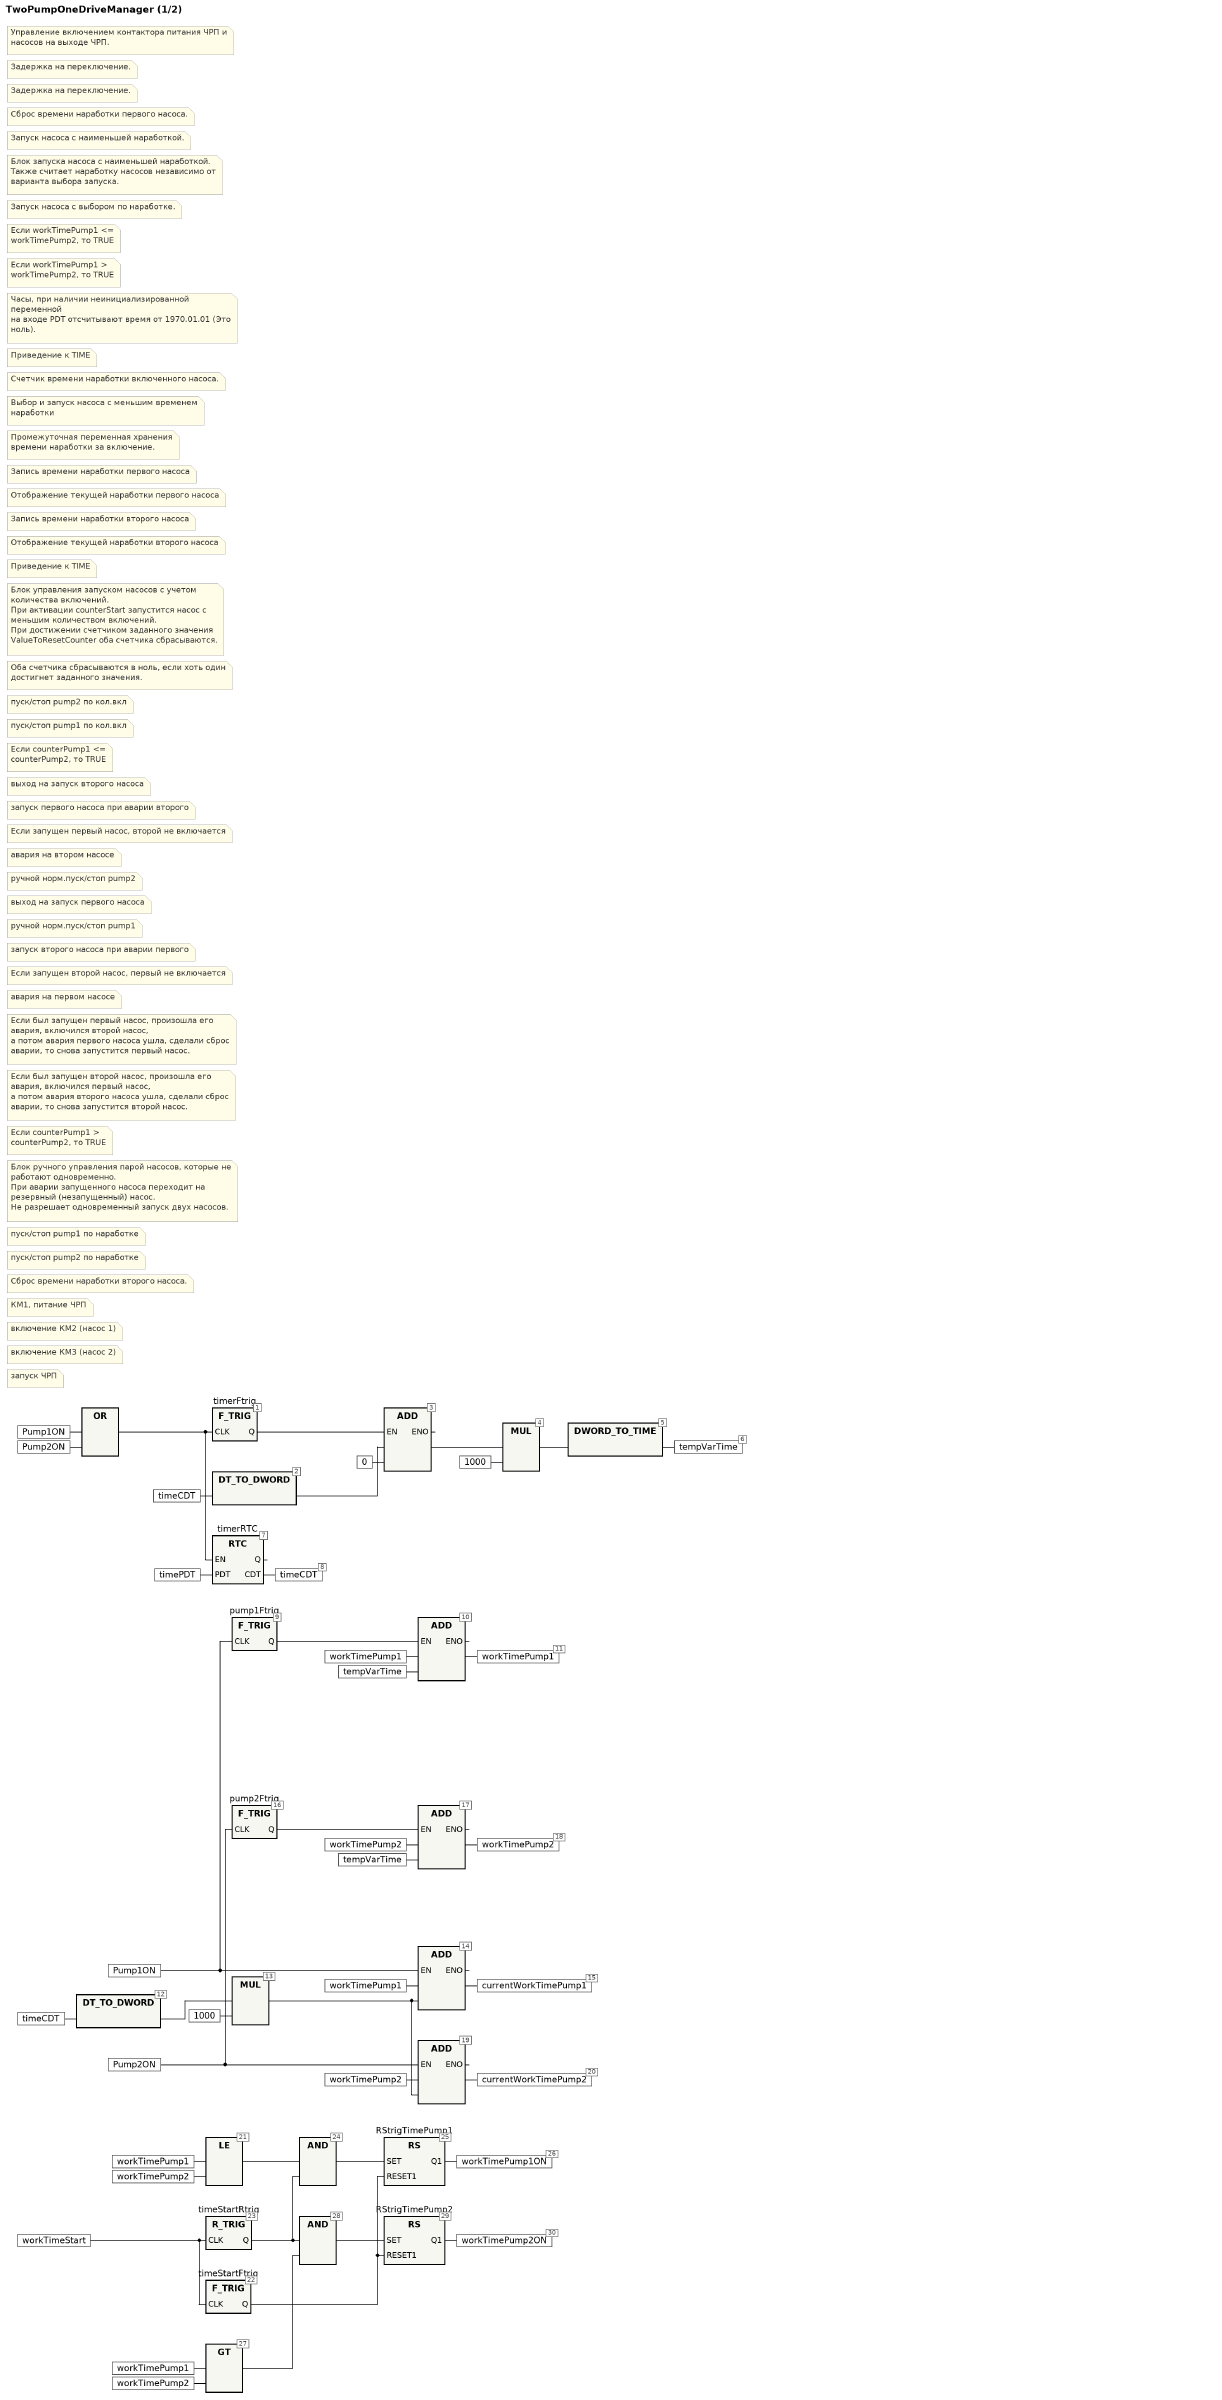
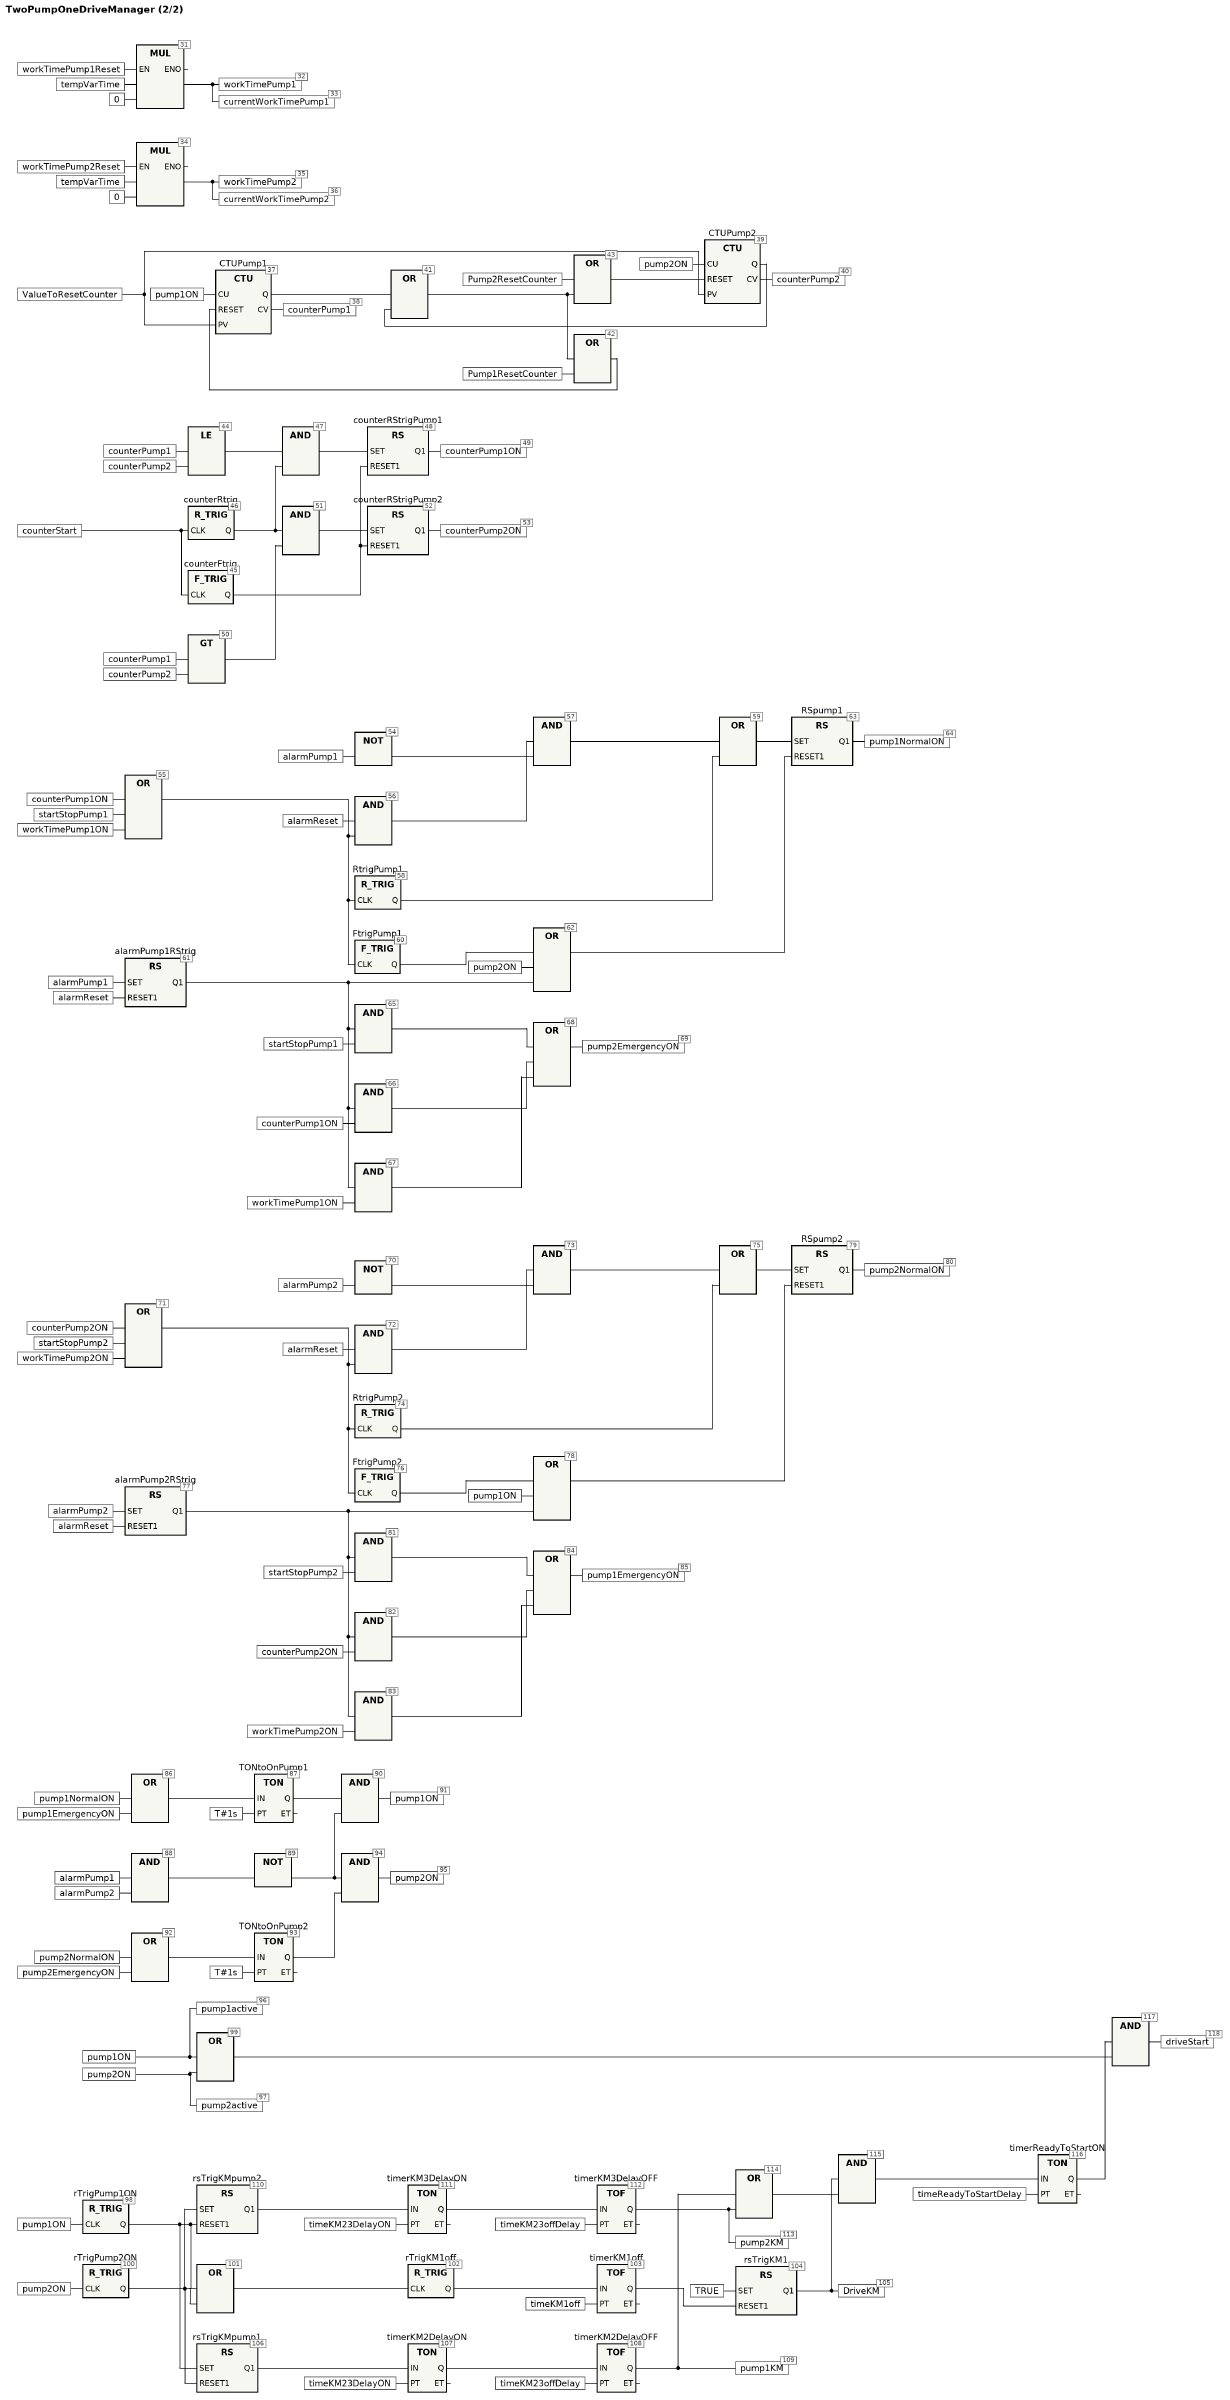
_CFC_ (* Continuous Function Chart, elements in execution order *)
(* Управление включением контактора питания ЧРП и насосов на выходе ЧРП. *)
(* Задержка на переключение. *)
(* Задержка на переключение. *)
(* Сброс времени наработки первого насоса. *)
(* Запуск насоса с наименьшей наработкой. *)
(* Блок запуска насоса с наименьшей наработкой. / Также считает наработку насосов независимо от варианта выбора запуска. *)
(* Запуск насоса с выбором по наработке. *)
(* Если workTimePump1 <= / workTimePump2, то TRUE *)
(* Если workTimePump1 > / workTimePump2, то TRUE *)
(* Часы, при наличии неинициализированной переменной / на входе PDT отсчитывают время от 1970.01.01 (Это ноль). *)
(* Приведение к TIME *)
(* Счетчик времени наработки включенного насоса. *)
(* Выбор и запуск насоса с меньшим временем наработки *)
(* Промежуточная переменная хранения / времени наработки за включение. *)
(* Запись времени наработки первого насоса *)
(* Отображение текущей наработки первого насоса *)
(* Запись времени наработки второго насоса *)
(* Отображение текущей наработки второго насоса *)
(* Приведение к TIME *)
(* Блок управления запуском насосов с учетом количества включений. / При активации counterStart запустится насос с меньшим количеством включений. / При достижении счетчиком заданного значения ValueToResetCounter оба счетчика сбрасываются. *)
(* Оба счетчика сбрасываются в ноль, если хоть один достигнет заданного значения. *)
(* пуск/стоп pump2 по кол.вкл *)
(* пуск/стоп pump1 по кол.вкл *)
(* Если counterPump1 <= / counterPump2, то TRUE *)
(* выход на запуск второго насоса *)
(* запуск первого насоса при аварии второго *)
(* Если запущен первый насос, второй не включается *)
(* авария на втором насосе *)
(* ручной норм.пуск/стоп pump2 *)
(* выход на запуск первого насоса *)
(* ручной норм.пуск/стоп pump1 *)
(* запуск второго насоса при аварии первого *)
(* Если запущен второй насос, первый не включается *)
(* авария на первом насосе *)
(* Если был запущен первый насос, произошла его авария, включился второй насос, / а потом авария первого насоса ушла, сделали сброс аварии, то снова запустится первый насос. *)
(* Если был запущен второй насос, произошла его авария, включился первый насос, / а потом авария второго насоса ушла, сделали сброс аварии, то снова запустится второй насос. *)
(* Если counterPump1 > / counterPump2, то TRUE *)
(* Блок ручного управления парой насосов, которые не работают одновременно. / При аварии запущенного насоса переходит на резервный (незапущенный) насос. / Не разрешает одновременный запуск двух насосов. *)
(* пуск/стоп pump1 по наработке *)
(* пуск/стоп pump2 по наработке *)
(* Сброс времени наработки второго насоса. *)
(* КМ1, питание ЧРП *)
(* включение КМ2 (насос 1) *)
(* включение КМ3 (насос 2) *)
(* запуск ЧРП *)
#0 OR(Pump1ON, Pump2ON)
#1 timerFtrig:F_TRIG(CLK: #0)
#2 DT_TO_DWORD(timeCDT)
#3 ADD(EN: #1.Q, #2, 0)
#4 MUL(#3, 1000)
#5 DWORD_TO_TIME(#4)
#6 tempVarTime <= #5
#7 timerRTC:RTC(EN: #0, PDT: timePDT)
#8 timeCDT <= #7.CDT
#9 pump1Ftrig:F_TRIG(CLK: Pump1ON)
#10 ADD(EN: #9.Q, workTimePump1, tempVarTime)
#11 workTimePump1 <= #10
#12 DT_TO_DWORD(timeCDT)
#13 MUL(#12, 1000)
#14 ADD(EN: Pump1ON, workTimePump1, #13)
#15 currentWorkTimePump1 <= #14
#16 pump2Ftrig:F_TRIG(CLK: Pump2ON)
#17 ADD(EN: #16.Q, workTimePump2, tempVarTime)
#18 workTimePump2 <= #17
#19 ADD(EN: Pump2ON, workTimePump2, #13)
#20 currentWorkTimePump2 <= #19
#21 LE(workTimePump1, workTimePump2)
#22 timeStartFtrig:F_TRIG(CLK: workTimeStart)
#23 timeStartRtrig:R_TRIG(CLK: workTimeStart)
#24 AND(#21, #23.Q)
#25 RStrigTimePump1:RS(SET: #24, RESET1: #22.Q)
#26 workTimePump1ON <= #25.Q1
#27 GT(workTimePump1, workTimePump2)
#28 AND(#23.Q, #27)
#29 RStrigTimePump2:RS(SET: #28, RESET1: #22.Q)
#30 workTimePump2ON <= #29.Q1
#31 MUL(EN: workTimePump1Reset, tempVarTime, 0)
#32 workTimePump1 <= #31
#33 currentWorkTimePump1 <= #31
#34 MUL(EN: workTimePump2Reset, tempVarTime, 0)
#35 workTimePump2 <= #34
#36 currentWorkTimePump2 <= #34
#37 CTUPump1:CTU(CU: pump1ON, RESET: #42, PV: ValueToResetCounter)
#38 counterPump1 <= #37.CV
#39 CTUPump2:CTU(CU: pump2ON, RESET: #43, PV: ValueToResetCounter)
#40 counterPump2 <= #39.CV
#41 OR(#37.Q, #39.Q)
#42 OR(#41, Pump1ResetCounter)
#43 OR(Pump2ResetCounter, #41)
#44 LE(counterPump1, counterPump2)
#45 counterFtrig:F_TRIG(CLK: counterStart)
#46 counterRtrig:R_TRIG(CLK: counterStart)
#47 AND(#44, #46.Q)
#48 counterRStrigPump1:RS(SET: #47, RESET1: #45.Q)
#49 counterPump1ON <= #48.Q1
#50 GT(counterPump1, counterPump2)
#51 AND(#46.Q, #50)
#52 counterRStrigPump2:RS(SET: #51, RESET1: #45.Q)
#53 counterPump2ON <= #52.Q1
#54 NOT(alarmPump1)
#55 OR(counterPump1ON, startStopPump1, workTimePump1ON)
#56 AND(alarmReset, #55)
#57 AND(#56, #54)
#58 RtrigPump1:R_TRIG(CLK: #55)
#59 OR(#57, #58.Q)
#60 FtrigPump1:F_TRIG(CLK: #55)
#61 alarmPump1RStrig:RS(SET: alarmPump1, RESET1: alarmReset)
#62 OR(#60.Q, pump2ON, #61.Q1)
#63 RSpump1:RS(SET: #59, RESET1: #62)
#64 pump1NormalON <= #63.Q1
#65 AND(#61.Q1, startStopPump1)
#66 AND(#61.Q1, counterPump1ON)
#67 AND(#61.Q1, workTimePump1ON)
#68 OR(#65, #66, #67)
#69 pump2EmergencyON <= #68
#70 NOT(alarmPump2)
#71 OR(counterPump2ON, startStopPump2, workTimePump2ON)
#72 AND(alarmReset, #71)
#73 AND(#72, #70)
#74 RtrigPump2:R_TRIG(CLK: #71)
#75 OR(#73, #74.Q)
#76 FtrigPump2:F_TRIG(CLK: #71)
#77 alarmPump2RStrig:RS(SET: alarmPump2, RESET1: alarmReset)
#78 OR(#76.Q, pump1ON, #77.Q1)
#79 RSpump2:RS(SET: #75, RESET1: #78)
#80 pump2NormalON <= #79.Q1
#81 AND(#77.Q1, startStopPump2)
#82 AND(#77.Q1, counterPump2ON)
#83 AND(#77.Q1, workTimePump2ON)
#84 OR(#81, #82, #83)
#85 pump1EmergencyON <= #84
#86 OR(pump1NormalON, pump1EmergencyON)
#87 TONtoOnPump1:TON(IN: #86, PT: T#1s)
#88 AND(alarmPump1, alarmPump2)
#89 NOT(#88)
#90 AND(#87.Q, #89)
#91 pump1ON <= #90
#92 OR(pump2NormalON, pump2EmergencyON)
#93 TONtoOnPump2:TON(IN: #92, PT: T#1s)
#94 AND(#89, #93.Q)
#95 pump2ON <= #94
#96 pump1active <= pump1ON
#97 pump2active <= pump2ON
#98 rTrigPump1ON:R_TRIG(CLK: pump1ON)
#99 OR(pump1ON, pump2ON)
#100 rTrigPump2ON:R_TRIG(CLK: pump2ON)
#101 OR(#98.Q, #100.Q)
#102 rTrigKM1off:R_TRIG(CLK: #101)
#103 timerKM1off:TOF(IN: #102.Q, PT: timeKM1off)
#104 rsTrigKM1:RS(SET: TRUE, RESET1: #103.Q)
#105 DriveKM <= #104.Q1
#106 rsTrigKMpump1:RS(SET: #98.Q, RESET1: #100.Q)
#107 timerKM2DelayON:TON(IN: #106.Q1, PT: timeKM23DelayON)
#108 timerKM2DelayOFF:TOF(IN: #107.Q, PT: timeKM23offDelay)
#109 pump1KM <= #108.Q
#110 rsTrigKMpump2:RS(SET: #100.Q, RESET1: #98.Q)
#111 timerKM3DelayON:TON(IN: #110.Q1, PT: timeKM23DelayON)
#112 timerKM3DelayOFF:TOF(IN: #111.Q, PT: timeKM23offDelay)
#113 pump2KM <= #112.Q
#114 OR(#108.Q, #112.Q)
#115 AND(#104.Q1, #114)
#116 timerReadyToStartON:TON(IN: #115, PT: timeReadyToStartDelay)
#117 AND(#116.Q, #99)
#118 driveStart <= #117
_END_CFC_
END_FUNCTION_BLOCK

(* POU SimpleValve, CFC *)
FUNCTION_BLOCK SimpleValve
VAR_INPUT
	inputOpen: BOOL;		(*вход подающий сигнал на открытие*)
	inputClose: BOOL;		(*вход, подающий сигнал на закрытие*)
	statusOpen: BOOL;		(*статус: заслонка/задвижка ОТКРЫТА*)
	statusClose: BOOL;		(*статус: заслонка/задвижка ЗАКРЫТА*)
	reset: BOOL;		(*ручной сброс выходов и аварий в неактивное состояние*)
	timeToOpenClose: TIME;		(*Время в секундах на открытие/закрытие (по тех.характеристикам прибора).*)
END_VAR
VAR_OUTPUT
	outputOpen: BOOL;		(*выход на открытие задвижки/заслонки*)
	outputClose: BOOL;		(*выход на закрытие задвижки/заслонки*)
	errorToOpen: BOOL;		(*авария на открытие - задвижка не открылась за заданное время.*)
	errorToClose: BOOL;		(*авария на закрытие - задвижка не закрылась за заданное время.*)
END_VAR
VAR
	toOpenTrigger: RS;
	toCloseTrigger: RS;
	timerToOpenClose: TON;
END_VAR
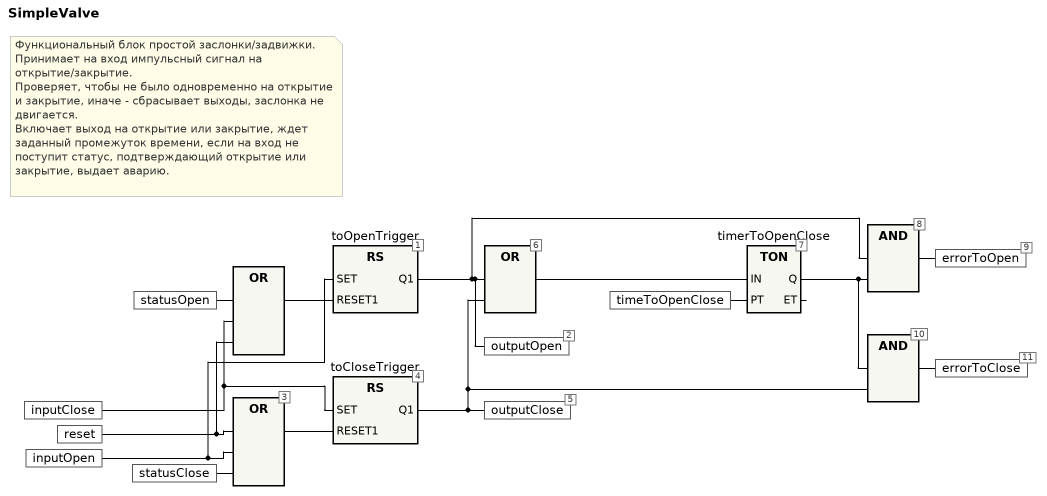
_CFC_ (* Continuous Function Chart, elements in execution order *)
(* Функциональный блок простой заслонки/задвижки. / Принимает на вход импульсный сигнал на открытие/закрытие. / Проверяет, чтобы не было одновременно на открытие и закрытие, иначе - сбрасывает выходы, заслонка не двигается. / Включает выход на открытие или закрытие, ждет заданный промежуток времени, если на вход не поступит статус, подтверждающий открытие или закрытие, выдает аварию. *)
#0 OR(statusOpen, inputClose, reset)
#1 toOpenTrigger:RS(SET: inputOpen, RESET1: #0)
#2 outputOpen <= #1.Q1
#3 OR(reset, inputOpen, statusClose)
#4 toCloseTrigger:RS(SET: inputClose, RESET1: #3)
#5 outputClose <= #4.Q1
#6 OR(#1.Q1, #4.Q1)
#7 timerToOpenClose:TON(IN: #6, PT: timeToOpenClose)
#8 AND(#1.Q1, #7.Q)
#9 errorToOpen <= #8
#10 AND(#7.Q, #4.Q1)
#11 errorToClose <= #10
_END_CFC_
(* the same logic as Structured Text *)
(* Функциональный блок простой заслонки/задвижки. / Принимает на вход импульсный сигнал на открытие/закрытие. / Проверяет, чтобы не было одновременно на открытие и закрытие, иначе - сбрасывает выходы, заслонка не двигается. / Включает выход на открытие или закрытие, ждет заданный промежуток времени, если на вход не поступит статус, подтверждающий открытие или закрытие, выдает аварию. *)
toOpenTrigger(SET := inputOpen, RESET1 := statusOpen OR inputClose OR reset);
outputOpen := toOpenTrigger.Q1;
toCloseTrigger(SET := inputClose, RESET1 := reset OR inputOpen OR statusClose);
outputClose := toCloseTrigger.Q1;
timerToOpenClose(IN := toOpenTrigger.Q1 OR toCloseTrigger.Q1, PT := timeToOpenClose);
errorToOpen := toOpenTrigger.Q1 AND timerToOpenClose.Q;
errorToClose := timerToOpenClose.Q AND toCloseTrigger.Q1;
END_FUNCTION_BLOCK

(* POU CounterTwoPumpManager, CFC *)
FUNCTION_BLOCK CounterTwoPumpManager
VAR_INPUT
	startStopPump1: BOOL;		(*Сигнал на пуск/стоп первого насоса.*)
	startStopPump2: BOOL;		(*Сигнал на пуск/стоп второго насоса.*)
	alarmPump1: BOOL;		(*Сигнал "авария" на первом насосе.*)
	alarmPump2: BOOL;		(*Сигнал "авария" на втором насосе.*)
	alarmReset: BOOL;		(*Сброс аварии.*)

	counterStart: BOOL;		(*Запуск насоса с меньшим количеством включений.*)
	Pump1ResetCounter: BOOL;		(*Сброс счетчика количества включений первого насоса. Сбрасывается также автоматически при достижении счетчиком значения ValueToResetCTU.*)
	Pump2ResetCounter: BOOL;		(*Сброс счетчика количества включений второго насоса. Сбрасывается также автоматически при достижении счетчиком значения ValueToResetCTU.*)
	ValueToResetCounter: WORD := 32767;		(*Значение счетчика, после которого он сбрасывается на ноль.
			Максимальное допустимое значение: 32767, будет установлено, если не подключать ничего на вход.*)
END_VAR
VAR_OUTPUT
	pump1ON: BOOL;		(*Выход на включение первого насоса.*)
	pump2ON: BOOL;		(*Выход на включение второго насоса.*)

	counterPump1: WORD;		(*Количество включений первого насоса. При достижении значения ValueToResetCTU сбрасывается в ноль.*)
	counterPump2: WORD;		(*Количество включений второго насоса. При достижении значения ValueToResetCTU сбрасывается в ноль.*)
END_VAR
VAR
	RtrigPump1: R_TRIG;		(*Включает первый насос по фронту сигнала на ручной пуск/стоп.*)
	FtrigPump1: F_TRIG;		(*Выключает первый насос по спаду сигнала на ручной пуск/стоп.*)
	RtrigPump2: R_TRIG;		(*Включает второй насос по фронту сигнала на ручной пуск/стоп.*)
	FtrigPump2: F_TRIG;		(*Выключает второй насос по спаду сигнала на ручной пуск/стоп.*)
	RSpump1: RS;		(*RS-триггер нормального включения первого насоса*)
	RSpump2: RS;		(*RS-триггер нормального включения второго насоса*)
	pump1NormalON: BOOL;		(*Сигнал нормального (неаварийного) включения первого насоса.*)
	pump2NormalON: BOOL;		(*Сигнал нормального (неаварийного) включения второго насоса.*)
	pump2EmergencyON: BOOL;		(*Сигнал аварийного включения второго насоса (при аварии первого).*)
	pump1EmergencyON: BOOL;		(*Сигнал аварийного включения первого насоса (при аварии второго).*)
	alarmPump1RStrig: RS;		(*Триггер аварии первого насоса.*)
	alarmPump2RStrig: RS;		(*Триггер аварии второго насоса.*)
	TONtoOnPump1: TON;		(*Таймер задержки включения первого насоса, на переключение контакторов при аварийном переключении.
			Жестко задано 1 секунда.*)
	TONtoOnPump2: TON;		(*Таймер задержки включения второго насоса, на переключение контакторов при аварийном переключении.
						Жестко задано 1 секунда.*)

	CTUPump1: CTU;		(*Счетчик количества включений первого насоса.*)
	CTUPump2: CTU;		(*Счетчик количества включений второго насоса.*)
	counterRtrig: R_TRIG;		(*Детектор переднего фронта сигнала на старт насоса с меньшей наработкой, включает насос.*)
	counterFtrig: F_TRIG;		(*Детектор спада сигнала на запуск насоса с меньшей наработкой, останавливает насос.*)
	counterRStrigPump1: RS;		(*Триггер-защелка включения первого насоса при запуске по количеству включений.*)
	counterRStrigPump2: RS;		(*Триггер-защелка включения второго насоса при запуске по количеству включений.*)
	counterPump1ON: BOOL;		(*Сигнал на запуск первого насоса при запуске по количеству включений.*)
	counterPump2ON: BOOL;		(*Сигнал на запуск второго насоса при запуске по количеству включений.*)

END_VAR
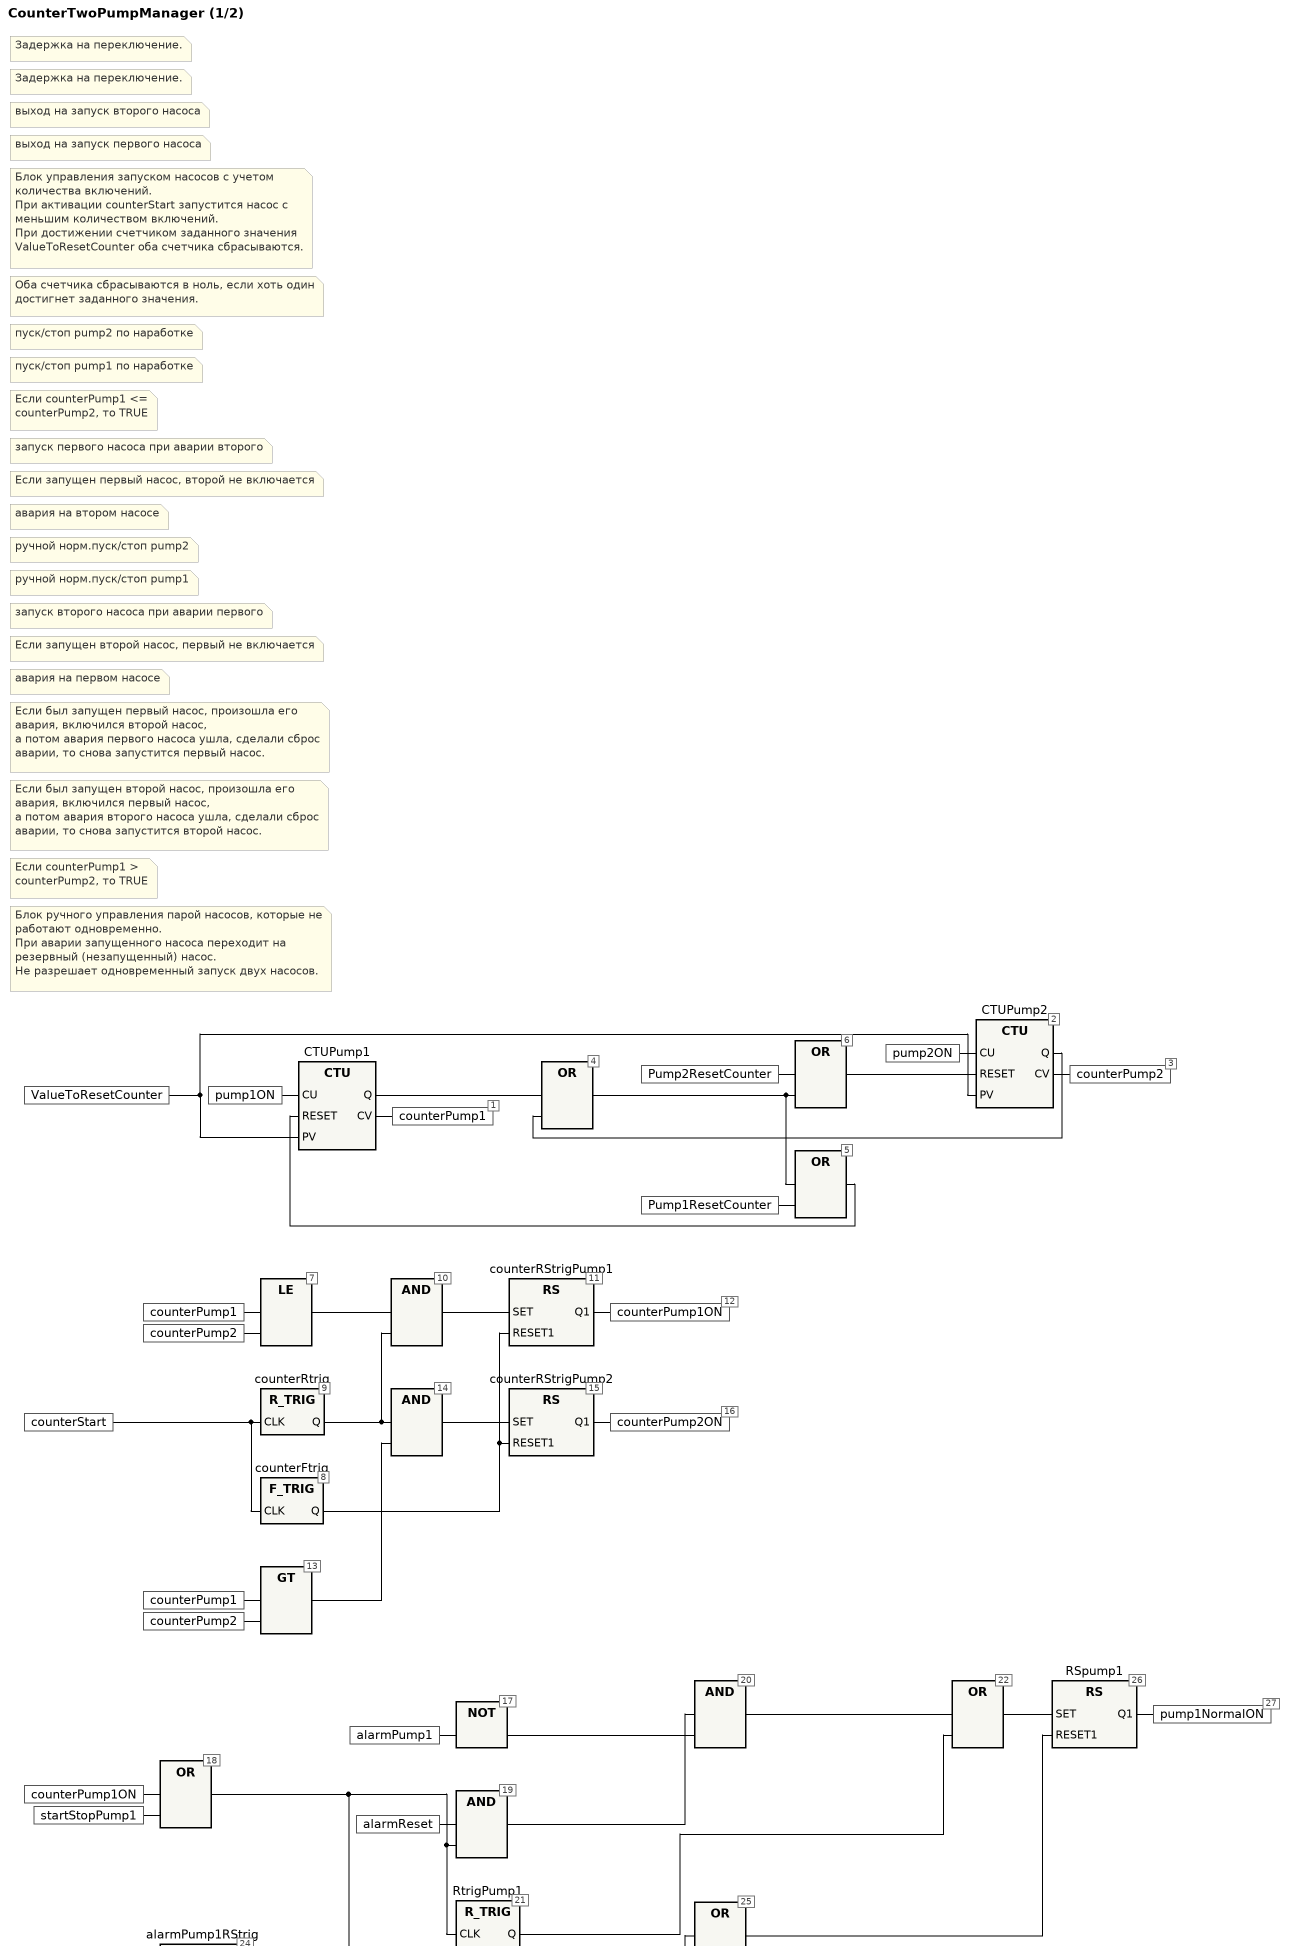
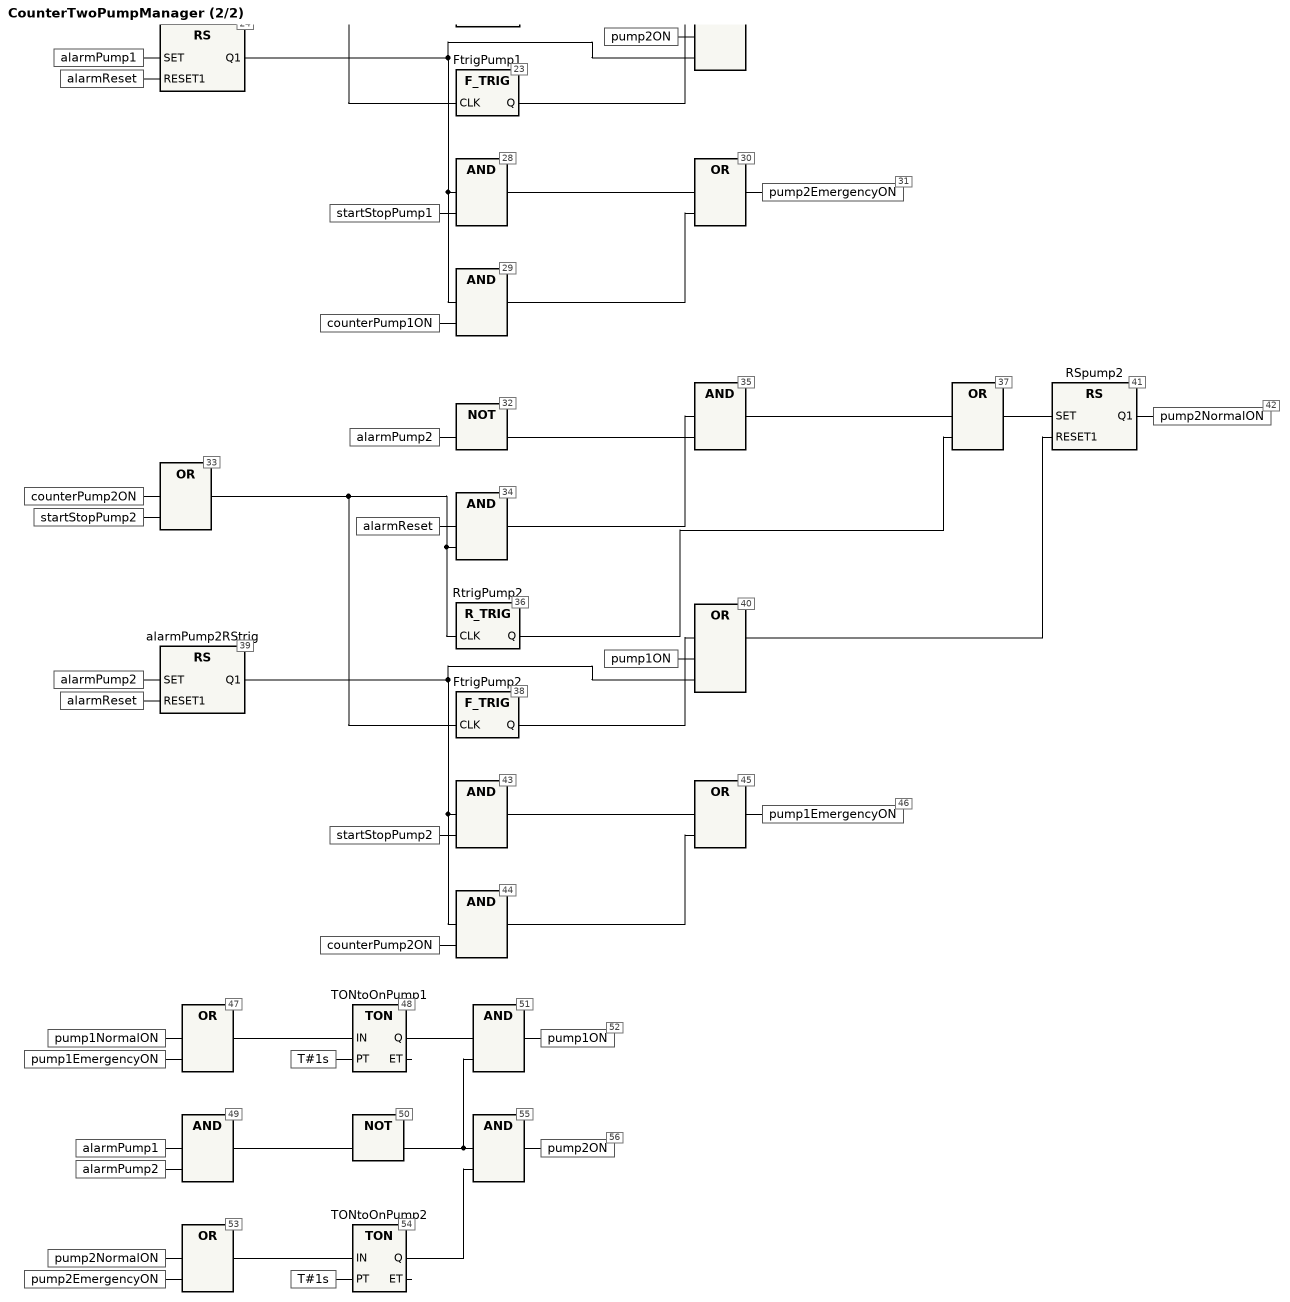
_CFC_ (* Continuous Function Chart, elements in execution order *)
(* Задержка на переключение. *)
(* Задержка на переключение. *)
(* выход на запуск второго насоса *)
(* выход на запуск первого насоса *)
(* Блок управления запуском насосов с учетом количества включений. / При активации counterStart запустится насос с меньшим количеством включений. / При достижении счетчиком заданного значения ValueToResetCounter оба счетчика сбрасываются. *)
(* Оба счетчика сбрасываются в ноль, если хоть один достигнет заданного значения. *)
(* пуск/стоп pump2 по наработке *)
(* пуск/стоп pump1 по наработке *)
(* Если counterPump1 <= / counterPump2, то TRUE *)
(* запуск первого насоса при аварии второго *)
(* Если запущен первый насос, второй не включается *)
(* авария на втором насосе *)
(* ручной норм.пуск/стоп pump2 *)
(* ручной норм.пуск/стоп pump1 *)
(* запуск второго насоса при аварии первого *)
(* Если запущен второй насос, первый не включается *)
(* авария на первом насосе *)
(* Если был запущен первый насос, произошла его авария, включился второй насос, / а потом авария первого насоса ушла, сделали сброс аварии, то снова запустится первый насос. *)
(* Если был запущен второй насос, произошла его авария, включился первый насос, / а потом авария второго насоса ушла, сделали сброс аварии, то снова запустится второй насос. *)
(* Если counterPump1 > / counterPump2, то TRUE *)
(* Блок ручного управления парой насосов, которые не работают одновременно. / При аварии запущенного насоса переходит на резервный (незапущенный) насос. / Не разрешает одновременный запуск двух насосов. *)
#0 CTUPump1:CTU(CU: pump1ON, RESET: #5, PV: ValueToResetCounter)
#1 counterPump1 <= #0.CV
#2 CTUPump2:CTU(CU: pump2ON, RESET: #6, PV: ValueToResetCounter)
#3 counterPump2 <= #2.CV
#4 OR(#0.Q, #2.Q)
#5 OR(#4, Pump1ResetCounter)
#6 OR(Pump2ResetCounter, #4)
#7 LE(counterPump1, counterPump2)
#8 counterFtrig:F_TRIG(CLK: counterStart)
#9 counterRtrig:R_TRIG(CLK: counterStart)
#10 AND(#7, #9.Q)
#11 counterRStrigPump1:RS(SET: #10, RESET1: #8.Q)
#12 counterPump1ON <= #11.Q1
#13 GT(counterPump1, counterPump2)
#14 AND(#9.Q, #13)
#15 counterRStrigPump2:RS(SET: #14, RESET1: #8.Q)
#16 counterPump2ON <= #15.Q1
#17 NOT(alarmPump1)
#18 OR(counterPump1ON, startStopPump1)
#19 AND(alarmReset, #18)
#20 AND(#19, #17)
#21 RtrigPump1:R_TRIG(CLK: #18)
#22 OR(#20, #21.Q)
#23 FtrigPump1:F_TRIG(CLK: #18)
#24 alarmPump1RStrig:RS(SET: alarmPump1, RESET1: alarmReset)
#25 OR(#23.Q, pump2ON, #24.Q1)
#26 RSpump1:RS(SET: #22, RESET1: #25)
#27 pump1NormalON <= #26.Q1
#28 AND(#24.Q1, startStopPump1)
#29 AND(#24.Q1, counterPump1ON)
#30 OR(#28, #29)
#31 pump2EmergencyON <= #30
#32 NOT(alarmPump2)
#33 OR(counterPump2ON, startStopPump2)
#34 AND(alarmReset, #33)
#35 AND(#34, #32)
#36 RtrigPump2:R_TRIG(CLK: #33)
#37 OR(#35, #36.Q)
#38 FtrigPump2:F_TRIG(CLK: #33)
#39 alarmPump2RStrig:RS(SET: alarmPump2, RESET1: alarmReset)
#40 OR(#38.Q, pump1ON, #39.Q1)
#41 RSpump2:RS(SET: #37, RESET1: #40)
#42 pump2NormalON <= #41.Q1
#43 AND(#39.Q1, startStopPump2)
#44 AND(#39.Q1, counterPump2ON)
#45 OR(#43, #44)
#46 pump1EmergencyON <= #45
#47 OR(pump1NormalON, pump1EmergencyON)
#48 TONtoOnPump1:TON(IN: #47, PT: T#1s)
#49 AND(alarmPump1, alarmPump2)
#50 NOT(#49)
#51 AND(#48.Q, #50)
#52 pump1ON <= #51
#53 OR(pump2NormalON, pump2EmergencyON)
#54 TONtoOnPump2:TON(IN: #53, PT: T#1s)
#55 AND(#50, #54.Q)
#56 pump2ON <= #55
_END_CFC_
END_FUNCTION_BLOCK

(* POU ImpulsCounter, CFC *)
FUNCTION_BLOCK ImpulsCounter
VAR_INPUT
	impulsInput: BOOL;		(*ходящие импульсы от расходомера.
			Каждый импульс будет прибавлять в итоговую сумму величину веса импульса.*)
	impulsValue: REAL;		(*Вес импульса расходомера.*)
	resetCounter: BOOL;		(*Сброс счетчика.*)
	correctionValue: REAL;		(*Число, которое будет прибавлено или вычтено из накопленной суммы.*)
	addCorrection: BOOL;		(*Прибавить коррекцию к накопленной сумме.*)
	deleteCorrection: BOOL;		(*Вычесть коррекцию из накопленной суммы.
			Если получится отрицательное число, сумма скинется в ноль.*)
END_VAR
VAR_OUTPUT
	totalAmountREAL: REAL;		(*Накопленная сумма в рациональном виде.
			В какой-то момент может выводится в экспоненциальной форме.*)
	totalAmountUDINT: UDINT;		(*Накопленная сумма в целочисленном виде.
			Округление десятичных по правилам арифметики.*)
END_VAR
VAR
	inputImpulsRtrig: R_TRIG;		(*Детектор переднего фронта входящих импульсов.*)
	resetRtrig: R_TRIG;		(*Детектор переднего фронта сигнала на сброс счетчика.*)
	addCorrRtrig: R_TRIG;		(*Детектор переднего фронта сигнала на прибавление коррекции.*)
	deleteCorrRtrig: R_TRIG;		(*Детектор переднего фронта сигнала на вычитание коррекции.*)
END_VAR
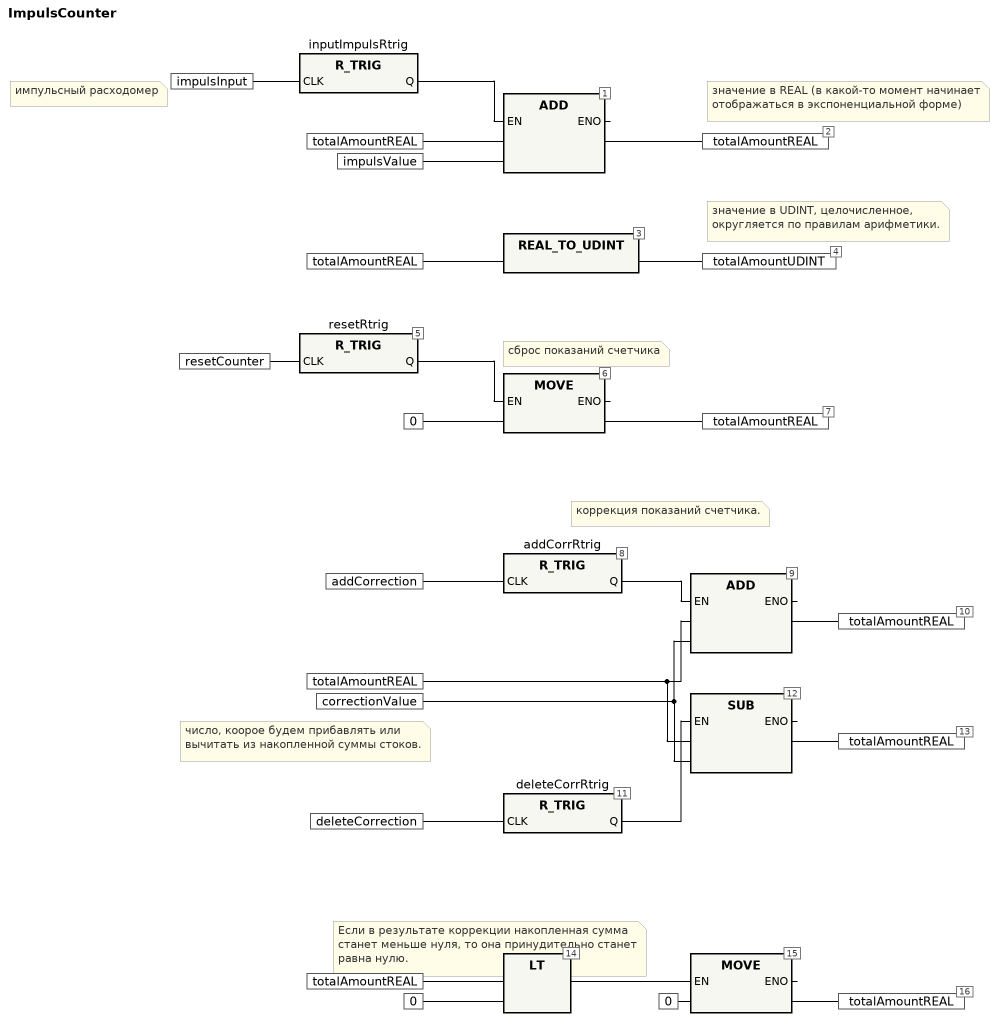
_CFC_ (* Continuous Function Chart, elements in execution order *)
(* импульсный расходомер *)
(* сброс показаний счетчика *)
(* значение в REAL (в какой-то момент начинает / отображаться в экспоненциальной форме) *)
(* значение в UDINT, целочисленное, / округляется по правилам арифметики. *)
(* Если в результате коррекции накопленная сумма станет меньше нуля, то она принудительно станет равна нулю. *)
(* коррекция показаний счетчика. *)
(* число, коорое будем прибавлять или / вычитать из накопленной суммы стоков. *)
#0 inputImpulsRtrig:R_TRIG(CLK: impulsInput)
#1 ADD(EN: #0.Q, totalAmountREAL, impulsValue)
#2 totalAmountREAL <= #1
#3 REAL_TO_UDINT(totalAmountREAL)
#4 totalAmountUDINT <= #3
#5 resetRtrig:R_TRIG(CLK: resetCounter)
#6 MOVE(EN: #5.Q, 0)
#7 totalAmountREAL <= #6
#8 addCorrRtrig:R_TRIG(CLK: addCorrection)
#9 ADD(EN: #8.Q, totalAmountREAL, correctionValue)
#10 totalAmountREAL <= #9
#11 deleteCorrRtrig:R_TRIG(CLK: deleteCorrection)
#12 SUB(EN: #11.Q, totalAmountREAL, correctionValue)
#13 totalAmountREAL <= #12
#14 LT(totalAmountREAL, 0)
#15 MOVE(EN: #14, 0)
#16 totalAmountREAL <= #15
_END_CFC_
(* the same logic as Structured Text *)
(* импульсный расходомер *)
(* сброс показаний счетчика *)
(* значение в REAL (в какой-то момент начинает / отображаться в экспоненциальной форме) *)
(* значение в UDINT, целочисленное, / округляется по правилам арифметики. *)
(* Если в результате коррекции накопленная сумма станет меньше нуля, то она принудительно станет равна нулю. *)
(* коррекция показаний счетчика. *)
(* число, коорое будем прибавлять или / вычитать из накопленной суммы стоков. *)
inputImpulsRtrig(CLK := impulsInput);
IF inputImpulsRtrig.Q THEN totalAmountREAL := totalAmountREAL + impulsValue; END_IF;
totalAmountUDINT := REAL_TO_UDINT(totalAmountREAL);
resetRtrig(CLK := resetCounter);
IF resetRtrig.Q THEN totalAmountREAL := 0; END_IF;
addCorrRtrig(CLK := addCorrection);
IF addCorrRtrig.Q THEN totalAmountREAL := totalAmountREAL + correctionValue; END_IF;
deleteCorrRtrig(CLK := deleteCorrection);
IF deleteCorrRtrig.Q THEN totalAmountREAL := totalAmountREAL - correctionValue; END_IF;
IF totalAmountREAL < 0 THEN totalAmountREAL := 0; END_IF;
END_FUNCTION_BLOCK

